LIN {X 0.280,Y -585.042,Z 449.322,A 0.000,B 0.000,C 90.000,E1 93.898} C_DIS
LIN {X -0.262,Y -588.278,Z 449.321,A 0.000,B 0.000,C 90.000,E1 93.841} C_DIS
LIN {X 0.026,Y -594.266,Z 449.320,A 0.000,B 0.000,C 90.000,E1 93.555} C_DIS
LIN {X 0.139,Y -599.956,Z 449.318,A 0.000,B 0.000,C 90.000,E1 93.212} C_DIS
LIN {X 0.002,Y -602.192,Z 449.317,A 0.000,B 0.000,C 90.000,E1 93.037} C_DIS
LIN {X -0.130,Y -605.915,Z 449.315,A 0.000,B 0.000,C 90.000,E1 92.694} C_DIS
LIN {X -0.222,Y -607.048,Z 449.314,A 0.000,B 0.000,C 90.000,E1 92.579} C_DIS
LIN {X 0.213,Y -608.066,Z 449.314,A 0.000,B 0.000,C 90.000,E1 92.407} C_DIS
LIN {X 0.153,Y -611.379,Z 449.311,A 0.000,B 0.000,C 90.000,E1 91.892} C_DIS
LIN {X 0.008,Y -612.023,Z 449.310,A 0.000,B 0.000,C 90.000,E1 91.776} C_DIS
LIN {X -0.029,Y -613.760,Z 449.307,A 0.000,B 0.000,C 90.000,E1 91.260} C_DIS
LIN {X -0.053,Y -614.433,Z 449.304,A 0.000,B 0.000,C 90.000,E1 90.745} C_DIS
LIN {X -0.069,Y -614.364,Z 449.301,A 0.000,B 0.000,C 90.000,E1 90.229} C_DIS
LIN {X 0.230,Y -614.158,Z 449.300,A 0.000,B 0.000,C 90.000,E1 89.943} C_DIS
LIN {X 0.214,Y -613.214,Z 449.297,A 0.000,B 0.000,C 90.000,E1 89.427} C_DIS
LIN {X -0.103,Y -612.227,Z 449.296,A 0.000,B 0.000,C 90.000,E1 89.198} C_DIS
LIN {X 0.030,Y -610.434,Z 449.293,A 0.000,B 0.000,C 90.000,E1 88.797} C_DIS
LIN {X -0.293,Y -608.948,Z 449.292,A 0.000,B 0.000,C 90.000,E1 88.568} C_DIS
LIN {X -0.015,Y -607.715,Z 449.290,A 0.000,B 0.000,C 90.000,E1 88.282} C_DIS
LIN {X 0.278,Y -606.083,Z 449.289,A 0.000,B 0.000,C 90.000,E1 87.993} C_DIS
LIN {X -0.227,Y -602.821,Z 449.287,A 0.000,B 0.000,C 90.000,E1 87.650} C_DIS
LIN {X 0.202,Y -601.337,Z 449.286,A 0.000,B 0.000,C 90.000,E1 87.478} C_DIS
LIN {X 0.029,Y -600.076,Z 449.285,A 0.000,B 0.000,C 90.000,E1 87.364} C_DIS
LIN {X 0.231,Y -595.856,Z 449.284,A 0.000,B 0.000,C 90.000,E1 87.020} C_DIS
LIN {X -0.293,Y -594.342,Z 449.283,A 0.000,B 0.000,C 90.000,E1 86.963} C_DIS
LIN {X -0.169,Y -592.394,Z 449.282,A 0.000,B 0.000,C 90.000,E1 86.846} C_DIS
LIN {X 0.126,Y -586.734,Z 449.281,A 0.000,B 0.000,C 90.000,E1 86.560} C_DIS
LIN {X 0.217,Y -581.356,Z 449.280,A 0.000,B 0.000,C 90.000,E1 86.331} C_DIS
LIN {X 0.124,Y -575.212,Z 449.279,A 0.000,B 0.000,C 90.000,E1 86.159} C_DIS
LIN {X -0.058,Y -574.482,Z 449.279,A 0.000,B 0.000,C 90.000,E1 86.159} C_DIS
LIN {X 0.129,Y -568.949,Z 449.278,A 0.000,B 0.000,C 90.000,E1 86.102} C_DIS
LIN {X 0.017,Y -568.335,Z 449.278,A 0.000,B 0.000,C 90.000,E1 86.102} C_DIS
LIN {X -0.038,Y -564.720,Z 449.278,A 0.000,B 0.000,C 90.000,E1 86.102} C_DIS
LIN {X -0.081,Y -486.304,Z 449.278,A 0.000,B 0.000,C 90.000,E1 86.102} C_DIS
LIN {X -0.033,Y -484.694,Z 449.254,A 0.000,B 0.000,C 90.000,E1 81.781} C_DIS
LIN {X -0.164,Y -484.577,Z 449.253,A 0.000,B 0.000,C 90.000,E1 81.489} C_DIS
LIN {X 0.184,Y -480.515,Z 449.227,A 0.000,B 0.000,C 90.000,E1 76.825} C_DIS
LIN {X 0.080,Y -474.266,Z 449.201,A 0.000,B 0.000,C 90.000,E1 72.181} C_DIS
LIN {X 0.048,Y -473.808,Z 449.199,A 0.000,B 0.000,C 90.000,E1 71.873} C_DIS
LIN {X 0.009,Y -466.228,Z 449.175,A 0.000,B 0.000,C 90.000,E1 67.486} C_DIS
LIN {X -0.049,Y -465.800,Z 449.173,A 0.000,B 0.000,C 90.000,E1 67.177} C_DIS
LIN {X 0.013,Y -464.449,Z 449.170,A 0.000,B 0.000,C 90.000,E1 66.538} C_DIS
LIN {X 0.209,Y -460.828,Z 449.160,A 0.000,B 0.000,C 90.000,E1 64.845} C_DIS
LIN {X 0.170,Y -460.829,Z 449.160,A 0.000,B 0.000,C 90.000,E1 64.845} C_DIS
LIN {X -0.103,Y -471.322,Z 449.152,A 0.000,B 0.000,C 90.000,E1 63.384} C_DIS
LIN {X -0.221,Y -476.895,Z 449.148,A 0.000,B 0.000,C 90.000,E1 62.615} C_DIS
LIN {X -0.218,Y -485.100,Z 449.141,A 0.000,B 0.000,C 90.000,E1 61.385} C_DIS
LIN {X 0.023,Y -489.694,Z 449.137,A 0.000,B 0.000,C 90.000,E1 60.589} C_DIS
LIN {X -0.151,Y -493.132,Z 449.133,A 0.000,B 0.000,C 90.000,E1 59.999} C_DIS
LIN {X -0.096,Y -495.546,Z 449.131,A 0.000,B 0.000,C 90.000,E1 59.537} C_DIS
LIN {X -0.176,Y -499.043,Z 449.127,A 0.000,B 0.000,C 90.000,E1 58.791} C_DIS
LIN {X -0.288,Y -501.495,Z 449.123,A 0.000,B 0.000,C 90.000,E1 58.201} C_DIS
LIN {X -0.118,Y -503.559,Z 449.120,A 0.000,B 0.000,C 90.000,E1 57.582} C_DIS
LIN {X -0.320,Y -506.063,Z 449.115,A 0.000,B 0.000,C 90.000,E1 56.707} C_DIS
LIN {X -0.116,Y -507.415,Z 449.112,A 0.000,B 0.000,C 90.000,E1 56.087} C_DIS
LIN {X 0.004,Y -508.918,Z 449.107,A 0.000,B 0.000,C 90.000,E1 55.182} C_DIS
LIN {X 0.139,Y -509.898,Z 449.102,A 0.000,B 0.000,C 90.000,E1 54.276} C_DIS
LIN {X -0.128,Y -510.426,Z 449.097,A 0.000,B 0.000,C 90.000,E1 53.417} C_DIS
LIN {X 0.242,Y -510.681,Z 449.090,A 0.000,B 0.000,C 90.000,E1 52.190} C_DIS
LIN {X 0.069,Y -510.714,Z 449.087,A 0.000,B 0.000,C 90.000,E1 51.618} C_DIS
LIN {X 0.040,Y -510.361,Z 449.080,A 0.000,B 0.000,C 90.000,E1 50.436} C_DIS
LIN {X 0.095,Y -509.924,Z 449.075,A 0.000,B 0.000,C 90.000,E1 49.542} C_DIS
LIN {X -0.099,Y -508.911,Z 449.067,A 0.000,B 0.000,C 90.000,E1 48.081} C_DIS
LIN {X -0.202,Y -507.992,Z 449.061,A 0.000,B 0.000,C 90.000,E1 46.905} C_DIS
LIN {X -0.318,Y -506.955,Z 449.054,A 0.000,B 0.000,C 90.000,E1 45.729} C_DIS
LIN {X -0.126,Y -505.056,Z 449.042,A 0.000,B 0.000,C 90.000,E1 43.623} C_DIS
LIN {X -0.190,Y -503.451,Z 449.032,A 0.000,B 0.000,C 90.000,E1 41.838} C_DIS
LIN {X -0.120,Y -502.051,Z 449.024,A 0.000,B 0.000,C 90.000,E1 40.334} C_DIS
LIN {X -0.076,Y -500.610,Z 449.016,A 0.000,B 0.000,C 90.000,E1 38.830} C_DIS
LIN {X 0.140,Y -499.520,Z 449.009,A 0.000,B 0.000,C 90.000,E1 37.604} C_DIS
LIN {X 0.083,Y -497.644,Z 448.999,A 0.000,B 0.000,C 90.000,E1 35.804} C_DIS
LIN {X 0.093,Y -495.608,Z 448.989,A 0.000,B 0.000,C 90.000,E1 33.992} C_DIS
LIN {X -0.070,Y -494.119,Z 448.982,A 0.000,B 0.000,C 90.000,E1 32.801} C_DIS
LIN {X -0.264,Y -491.817,Z 448.972,A 0.000,B 0.000,C 90.000,E1 31.003} C_DIS
LIN {X 0.091,Y -490.273,Z 448.965,A 0.000,B 0.000,C 90.000,E1 29.745} C_DIS
LIN {X -0.186,Y -487.521,Z 448.953,A 0.000,B 0.000,C 90.000,E1 27.641} C_DIS
LIN {X 0.105,Y -484.639,Z 448.940,A 0.000,B 0.000,C 90.000,E1 25.155} C_DIS
LIN {X 0.102,Y -481.751,Z 448.923,A 0.000,B 0.000,C 90.000,E1 22.078} C_DIS
LIN {X -0.089,Y -480.184,Z 448.911,A 0.000,B 0.000,C 90.000,E1 19.939} C_DIS
LIN {X 0.145,Y -479.024,Z 448.900,A 0.000,B 0.000,C 90.000,E1 18.055} C_DIS
LIN {X 0.056,Y -477.797,Z 448.890,A 0.000,B 0.000,C 90.000,E1 16.205} C_DIS
LIN {X -0.020,Y -476.715,Z 448.882,A 0.000,B 0.000,C 90.000,E1 14.662} C_DIS
LIN {X -0.033,Y -475.299,Z 448.868,A 0.000,B 0.000,C 90.000,E1 12.175} C_DIS
LIN {X 0.065,Y -474.352,Z 448.854,A 0.000,B 0.000,C 90.000,E1 9.670} C_DIS
LIN {X -0.039,Y -474.103,Z 448.849,A 0.000,B 0.000,C 90.000,E1 8.746} C_DIS
LIN {X -0.156,Y -473.933,Z 448.826,A 0.000,B 0.000,C 90.000,E1 4.702} C_DIS
LIN {X -0.023,Y -475.423,Z 448.804,A 0.000,B 0.000,C 90.000,E1 0.630} C_DIS
LIN {X -0.013,Y -477.940,Z 448.785,A 0.000,B 0.000,C 90.000,E1 357.306} C_DIS
LIN {X -0.097,Y -480.676,Z 448.771,A 0.000,B 0.000,C 90.000,E1 354.837} C_DIS
LIN {X 0.000,Y -483.958,Z 448.758,A 0.000,B 0.000,C 90.000,E1 352.356} C_DIS
LIN {X -0.018,Y -487.182,Z 448.746,A 0.000,B 0.000,C 90.000,E1 350.208} C_DIS
LIN {X -0.090,Y -495.576,Z 448.720,A 0.000,B 0.000,C 90.000,E1 345.644} C_DIS
LIN {X 0.146,Y -500.335,Z 448.708,A 0.000,B 0.000,C 90.000,E1 343.504} C_DIS
LIN {X -0.300,Y -506.989,Z 448.694,A 0.000,B 0.000,C 90.000,E1 340.859} C_DIS
LIN {X 0.233,Y -512.497,Z 448.682,A 0.000,B 0.000,C 90.000,E1 338.720} C_DIS
LIN {X -0.111,Y -516.460,Z 448.674,A 0.000,B 0.000,C 90.000,E1 337.283} C_DIS
LIN {X -0.087,Y -521.973,Z 448.662,A 0.000,B 0.000,C 90.000,E1 335.229} C_DIS
LIN {X 0.117,Y -526.692,Z 448.653,A 0.000,B 0.000,C 90.000,E1 333.461} C_DIS
LIN {X 0.014,Y -530.575,Z 448.645,A 0.000,B 0.000,C 90.000,E1 332.025} C_DIS
LIN {X -0.300,Y -535.330,Z 448.635,A 0.000,B 0.000,C 90.000,E1 330.333} C_DIS
LIN {X -0.153,Y -537.751,Z 448.630,A 0.000,B 0.000,C 90.000,E1 329.459} C_DIS
LIN {X -0.056,Y -542.540,Z 448.621,A 0.000,B 0.000,C 90.000,E1 327.740} C_DIS
LIN {X 0.228,Y -546.447,Z 448.613,A 0.000,B 0.000,C 90.000,E1 326.294} C_DIS
LIN {X 0.137,Y -550.354,Z 448.605,A 0.000,B 0.000,C 90.000,E1 324.895} C_DIS
LIN {X -0.111,Y -556.790,Z 448.593,A 0.000,B 0.000,C 90.000,E1 322.683} C_DIS
LIN {X 0.156,Y -563.379,Z 448.580,A 0.000,B 0.000,C 90.000,E1 320.436} C_DIS
LIN {X 0.295,Y -568.567,Z 448.571,A 0.000,B 0.000,C 90.000,E1 318.771} C_DIS
LIN {X -0.004,Y -572.710,Z 448.564,A 0.000,B 0.000,C 90.000,E1 317.433} C_DIS
LIN {X -0.096,Y -577.611,Z 448.555,A 0.000,B 0.000,C 90.000,E1 315.810} C_DIS
LIN {X -0.107,Y -582.531,Z 448.546,A 0.000,B 0.000,C 90.000,E1 314.190} C_DIS
LIN {X 0.151,Y -588.401,Z 448.535,A 0.000,B 0.000,C 90.000,E1 312.285} C_DIS
LIN {X -0.210,Y -592.519,Z 448.528,A 0.000,B 0.000,C 90.000,E1 310.987} C_DIS
LIN {X -0.049,Y -596.549,Z 448.520,A 0.000,B 0.000,C 90.000,E1 309.644} C_DIS
LIN {X 0.052,Y -601.175,Z 448.511,A 0.000,B 0.000,C 90.000,E1 308.051} C_DIS
LIN {X -0.006,Y -604.976,Z 448.504,A 0.000,B 0.000,C 90.000,E1 306.744} C_DIS
LIN {X -0.012,Y -608.601,Z 448.497,A 0.000,B 0.000,C 90.000,E1 305.438} C_DIS
LIN {X -0.035,Y -610.772,Z 448.493,A 0.000,B 0.000,C 90.000,E1 304.659} C_DIS
LIN {X -0.149,Y -614.195,Z 448.485,A 0.000,B 0.000,C 90.000,E1 303.372} C_DIS
LIN {X 0.104,Y -618.070,Z 448.477,A 0.000,B 0.000,C 90.000,E1 301.799} C_DIS
LIN {X 0.104,Y -621.763,Z 448.468,A 0.000,B 0.000,C 90.000,E1 300.256} C_DIS
LIN {X -0.144,Y -624.574,Z 448.461,A 0.000,B 0.000,C 90.000,E1 298.999} C_DIS
LIN {X -0.056,Y -628.494,Z 448.451,A 0.000,B 0.000,C 90.000,E1 297.206} C_DIS
LIN {X 0.044,Y -630.613,Z 448.446,A 0.000,B 0.000,C 90.000,E1 296.181} C_DIS
LIN {X 0.205,Y -633.127,Z 448.438,A 0.000,B 0.000,C 90.000,E1 294.899} C_DIS
LIN {X 0.176,Y -635.790,Z 448.430,A 0.000,B 0.000,C 90.000,E1 293.387} C_DIS
LIN {X -0.058,Y -638.246,Z 448.422,A 0.000,B 0.000,C 90.000,E1 291.897} C_DIS
LIN {X 0.299,Y -640.073,Z 448.415,A 0.000,B 0.000,C 90.000,E1 290.610} C_DIS
LIN {X 0.038,Y -641.527,Z 448.409,A 0.000,B 0.000,C 90.000,E1 289.631} C_DIS
LIN {X -0.212,Y -642.795,Z 448.404,A 0.000,B 0.000,C 90.000,E1 288.652} C_DIS
LIN {X -0.196,Y -644.148,Z 448.397,A 0.000,B 0.000,C 90.000,E1 287.402} C_DIS
LIN {X -0.111,Y -645.549,Z 448.388,A 0.000,B 0.000,C 90.000,E1 285.898} C_DIS
LIN {X -0.066,Y -646.361,Z 448.383,A 0.000,B 0.000,C 90.000,E1 284.898} C_DIS
LIN {X 0.015,Y -647.149,Z 448.376,A 0.000,B 0.000,C 90.000,E1 283.647} C_DIS
LIN {X 0.085,Y -647.640,Z 448.370,A 0.000,B 0.000,C 90.000,E1 282.647} C_DIS
LIN {X -0.112,Y -648.117,Z 448.363,A 0.000,B 0.000,C 90.000,E1 281.422} C_DIS
LIN {X -0.038,Y -648.313,Z 448.358,A 0.000,B 0.000,C 90.000,E1 280.423} C_DIS
LIN {X -0.338,Y -648.217,Z 448.351,A 0.000,B 0.000,C 90.000,E1 279.208} C_DIS
LIN {X -0.237,Y -648.029,Z 448.347,A 0.000,B 0.000,C 90.000,E1 278.454} C_DIS
LIN {X 0.110,Y -647.485,Z 448.340,A 0.000,B 0.000,C 90.000,E1 277.182} C_DIS
LIN {X 0.197,Y -647.015,Z 448.336,A 0.000,B 0.000,C 90.000,E1 276.429} C_DIS
LIN {X 0.205,Y -646.363,Z 448.332,A 0.000,B 0.000,C 90.000,E1 275.682} C_DIS
LIN {X 0.036,Y -645.158,Z 448.326,A 0.000,B 0.000,C 90.000,E1 274.702} C_DIS
LIN {X 0.028,Y -644.107,Z 448.322,A 0.000,B 0.000,C 90.000,E1 273.955} C_DIS
LIN {X -0.228,Y -642.506,Z 448.316,A 0.000,B 0.000,C 90.000,E1 272.980} C_DIS
LIN {X -0.104,Y -640.224,Z 448.310,A 0.000,B 0.000,C 90.000,E1 271.718} C_DIS
LIN {X 0.209,Y -638.223,Z 448.304,A 0.000,B 0.000,C 90.000,E1 270.688} C_DIS
LIN {X -0.004,Y -634.937,Z 448.296,A 0.000,B 0.000,C 90.000,E1 269.198} C_DIS
LIN {X 0.235,Y -632.504,Z 448.290,A 0.000,B 0.000,C 90.000,E1 268.167} C_DIS
LIN {X 0.185,Y -629.317,Z 448.283,A 0.000,B 0.000,C 90.000,E1 266.906} C_DIS
LIN {X -0.161,Y -625.337,Z 448.274,A 0.000,B 0.000,C 90.000,E1 265.412} C_DIS
LIN {X 0.098,Y -621.272,Z 448.266,A 0.000,B 0.000,C 90.000,E1 263.856} C_DIS
LIN {X 0.227,Y -618.487,Z 448.260,A 0.000,B 0.000,C 90.000,E1 262.818} C_DIS
LIN {X -0.181,Y -614.200,Z 448.252,A 0.000,B 0.000,C 90.000,E1 261.310} C_DIS
LIN {X 0.186,Y -610.466,Z 448.245,A 0.000,B 0.000,C 90.000,E1 259.982} C_DIS
LIN {X -0.020,Y -606.615,Z 448.237,A 0.000,B 0.000,C 90.000,E1 258.701} C_DIS
LIN {X -0.169,Y -602.656,Z 448.230,A 0.000,B 0.000,C 90.000,E1 257.409} C_DIS
LIN {X 0.202,Y -598.611,Z 448.223,A 0.000,B 0.000,C 90.000,E1 256.061} C_DIS
LIN {X 0.070,Y -596.121,Z 448.218,A 0.000,B 0.000,C 90.000,E1 255.283} C_DIS
LIN {X -0.104,Y -591.867,Z 448.211,A 0.000,B 0.000,C 90.000,E1 253.976} C_DIS
LIN {X -0.182,Y -587.539,Z 448.204,A 0.000,B 0.000,C 90.000,E1 252.653} C_DIS
LIN {X 0.222,Y -583.092,Z 448.196,A 0.000,B 0.000,C 90.000,E1 251.275} C_DIS
LIN {X -0.212,Y -579.432,Z 448.190,A 0.000,B 0.000,C 90.000,E1 250.242} C_DIS
LIN {X 0.048,Y -575.781,Z 448.184,A 0.000,B 0.000,C 90.000,E1 249.135} C_DIS
LIN {X -0.126,Y -570.969,Z 448.177,A 0.000,B 0.000,C 90.000,E1 247.794} C_DIS
LIN {X 0.227,Y -566.950,Z 448.171,A 0.000,B 0.000,C 90.000,E1 246.666} C_DIS
LIN {X 0.098,Y -561.760,Z 448.163,A 0.000,B 0.000,C 90.000,E1 245.305} C_DIS
LIN {X 0.131,Y -555.431,Z 448.154,A 0.000,B 0.000,C 90.000,E1 243.640} C_DIS
LIN {X 0.033,Y -549.002,Z 448.144,A 0.000,B 0.000,C 90.000,E1 241.975} C_DIS
LIN {X 0.059,Y -541.652,Z 448.133,A 0.000,B 0.000,C 90.000,E1 239.999} C_DIS
LIN {X 0.177,Y -534.469,Z 448.122,A 0.000,B 0.000,C 90.000,E1 237.995} C_DIS
LIN {X -0.032,Y -528.228,Z 448.113,A 0.000,B 0.000,C 90.000,E1 236.294} C_DIS
LIN {X -0.084,Y -522.049,Z 448.103,A 0.000,B 0.000,C 90.000,E1 234.562} C_DIS
LIN {X 0.271,Y -514.861,Z 448.092,A 0.000,B 0.000,C 90.000,E1 232.477} C_DIS
LIN {X 0.068,Y -505.494,Z 448.075,A 0.000,B 0.000,C 90.000,E1 229.542} C_DIS
LIN {X -0.217,Y -501.066,Z 448.067,A 0.000,B 0.000,C 90.000,E1 228.081} C_DIS
LIN {X 0.123,Y -496.709,Z 448.059,A 0.000,B 0.000,C 90.000,E1 226.539} C_DIS
LIN {X 0.184,Y -489.920,Z 448.045,A 0.000,B 0.000,C 90.000,E1 224.109} C_DIS
LIN {X 0.100,Y -485.033,Z 448.035,A 0.000,B 0.000,C 90.000,E1 222.285} C_DIS
LIN {X -0.061,Y -480.269,Z 448.025,A 0.000,B 0.000,C 90.000,E1 220.458} C_DIS
LIN {X -0.172,Y -474.944,Z 448.013,A 0.000,B 0.000,C 90.000,E1 218.302} C_DIS
LIN {X -0.034,Y -468.523,Z 447.997,A 0.000,B 0.000,C 90.000,E1 215.471} C_DIS
LIN {X -0.023,Y -464.476,Z 447.987,A 0.000,B 0.000,C 90.000,E1 213.579} C_DIS
LIN {X -0.122,Y -459.209,Z 447.972,A 0.000,B 0.000,C 90.000,E1 211.052} C_DIS
LIN {X -0.165,Y -456.005,Z 447.964,A 0.000,B 0.000,C 90.000,E1 209.461} C_DIS
LIN {X -0.090,Y -452.779,Z 447.955,A 0.000,B 0.000,C 90.000,E1 207.847} C_DIS
LIN {X -0.074,Y -449.527,Z 447.946,A 0.000,B 0.000,C 90.000,E1 206.232} C_DIS
LIN {X 0.000,Y -444.815,Z 447.933,A 0.000,B 0.000,C 90.000,E1 203.951} C_DIS
LIN {X 0.147,Y -440.894,Z 447.922,A 0.000,B 0.000,C 90.000,E1 201.972} C_DIS
LIN {X 0.032,Y -436.381,Z 447.909,A 0.000,B 0.000,C 90.000,E1 199.685} C_DIS
LIN {X -0.005,Y -431.687,Z 447.895,A 0.000,B 0.000,C 90.000,E1 197.040} C_DIS
LIN {X 0.223,Y -428.444,Z 447.884,A 0.000,B 0.000,C 90.000,E1 195.009} C_DIS
LIN {X -0.077,Y -424.908,Z 447.871,A 0.000,B 0.000,C 90.000,E1 192.703} C_DIS
LIN {X -0.023,Y -420.328,Z 447.852,A 0.000,B 0.000,C 90.000,E1 189.321} C_DIS
LIN {X -0.100,Y -417.898,Z 447.841,A 0.000,B 0.000,C 90.000,E1 187.296} C_DIS
LIN {X 0.179,Y -415.008,Z 447.825,A 0.000,B 0.000,C 90.000,E1 184.531} C_DIS
LIN {X -0.133,Y -412.454,Z 447.810,A 0.000,B 0.000,C 90.000,E1 181.835} C_DIS
LIN {X -0.124,Y -410.004,Z 447.789,A 0.000,B 0.000,C 90.000,E1 178.051} C_DIS
LIN {X -0.144,Y -408.668,Z 447.766,A 0.000,B 0.000,C 90.000,E1 173.913} C_DIS
LIN {X -0.059,Y -408.839,Z 447.749,A 0.000,B 0.000,C 90.000,E1 170.792} C_DIS
LIN {X -0.040,Y -410.037,Z 447.728,A 0.000,B 0.000,C 90.000,E1 166.992} C_DIS
LIN {X -0.110,Y -412.024,Z 447.709,A 0.000,B 0.000,C 90.000,E1 163.559} C_DIS
LIN {X -0.013,Y -415.002,Z 447.690,A 0.000,B 0.000,C 90.000,E1 160.115} C_DIS
LIN {X 0.099,Y -417.197,Z 447.678,A 0.000,B 0.000,C 90.000,E1 158.050} C_DIS
LIN {X 0.223,Y -421.074,Z 447.661,A 0.000,B 0.000,C 90.000,E1 154.973} C_DIS
LIN {X 0.158,Y -424.385,Z 447.648,A 0.000,B 0.000,C 90.000,E1 152.615} C_DIS
LIN {X 0.204,Y -427.985,Z 447.635,A 0.000,B 0.000,C 90.000,E1 150.255} C_DIS
LIN {X -0.033,Y -430.105,Z 447.628,A 0.000,B 0.000,C 90.000,E1 148.948} C_DIS
LIN {X -0.100,Y -435.215,Z 447.611,A 0.000,B 0.000,C 90.000,E1 145.960} C_DIS
LIN {X 0.110,Y -440.091,Z 447.596,A 0.000,B 0.000,C 90.000,E1 143.290} C_DIS
LIN {X 0.052,Y -442.701,Z 447.589,A 0.000,B 0.000,C 90.000,E1 141.984} C_DIS
LIN {X 0.006,Y -446.040,Z 447.580,A 0.000,B 0.000,C 90.000,E1 140.356} C_DIS
LIN {X 0.020,Y -449.451,Z 447.571,A 0.000,B 0.000,C 90.000,E1 138.728} C_DIS
LIN {X -0.286,Y -452.143,Z 447.564,A 0.000,B 0.000,C 90.000,E1 137.472} C_DIS
LIN {X 0.113,Y -455.291,Z 447.555,A 0.000,B 0.000,C 90.000,E1 135.810} C_DIS
LIN {X 0.188,Y -456.958,Z 447.549,A 0.000,B 0.000,C 90.000,E1 134.838} C_DIS
LIN {X 0.283,Y -458.534,Z 447.544,A 0.000,B 0.000,C 90.000,E1 133.866} C_DIS
LIN {X 0.117,Y -460.215,Z 447.537,A 0.000,B 0.000,C 90.000,E1 132.609} C_DIS
LIN {X -0.028,Y -461.379,Z 447.530,A 0.000,B 0.000,C 90.000,E1 131.353} C_DIS
LIN {X 0.142,Y -461.921,Z 447.524,A 0.000,B 0.000,C 90.000,E1 130.378} C_DIS
LIN {X 0.025,Y -461.985,Z 447.519,A 0.000,B 0.000,C 90.000,E1 129.439} C_DIS
LIN {X -0.190,Y -461.777,Z 447.516,A 0.000,B 0.000,C 90.000,E1 128.830} C_DIS
LIN {X -0.019,Y -461.057,Z 447.510,A 0.000,B 0.000,C 90.000,E1 127.855} C_DIS
LIN {X 0.225,Y -459.977,Z 447.505,A 0.000,B 0.000,C 90.000,E1 126.870} C_DIS
LIN {X 0.079,Y -459.118,Z 447.501,A 0.000,B 0.000,C 90.000,E1 126.251} C_DIS
LIN {X 0.200,Y -458.102,Z 447.498,A 0.000,B 0.000,C 90.000,E1 125.598} C_DIS
LIN {X 0.038,Y -456.132,Z 447.493,A 0.000,B 0.000,C 90.000,E1 124.659} C_DIS
LIN {X -0.132,Y -454.724,Z 447.489,A 0.000,B 0.000,C 90.000,E1 124.040} C_DIS
LIN {X -0.123,Y -451.310,Z 447.482,A 0.000,B 0.000,C 90.000,E1 122.752} C_DIS
LIN {X 0.139,Y -448.558,Z 447.477,A 0.000,B 0.000,C 90.000,E1 121.750} C_DIS
LIN {X -0.013,Y -445.715,Z 447.471,A 0.000,B 0.000,C 90.000,E1 120.797} C_DIS
LIN {X 0.069,Y -440.549,Z 447.462,A 0.000,B 0.000,C 90.000,E1 119.155} C_DIS
LIN {X 0.105,Y -436.433,Z 447.455,A 0.000,B 0.000,C 90.000,E1 117.897} C_DIS
LIN {X 0.066,Y -436.421,Z 447.455,A 0.000,B 0.000,C 90.000,E1 117.897} C_DIS
LIN {X -0.083,Y -444.882,Z 447.438,A 0.000,B 0.000,C 90.000,E1 114.899} C_DIS
LIN {X 0.176,Y -453.993,Z 447.417,A 0.000,B 0.000,C 90.000,E1 110.972} C_DIS
LIN {X 0.288,Y -456.641,Z 447.411,A 0.000,B 0.000,C 90.000,E1 109.993} C_DIS
LIN {X 0.035,Y -457.454,Z 447.410,A 0.000,B 0.000,C 90.000,E1 109.704} C_DIS
LIN {X 0.136,Y -466.113,Z 447.387,A 0.000,B 0.000,C 90.000,E1 105.552} C_DIS
LIN {X -0.140,Y -467.684,Z 447.383,A 0.000,B 0.000,C 90.000,E1 104.954} C_DIS
LIN {X -0.183,Y -475.897,Z 447.357,A 0.000,B 0.000,C 90.000,E1 100.254} C_DIS
LIN {X 0.124,Y -476.347,Z 447.355,A 0.000,B 0.000,C 90.000,E1 99.905} C_DIS
LIN {X 0.081,Y -481.861,Z 447.331,A 0.000,B 0.000,C 90.000,E1 95.568} C_DIS
LIN {X -0.072,Y -482.189,Z 447.329,A 0.000,B 0.000,C 90.000,E1 95.277} C_DIS
LIN {X -0.196,Y -483.242,Z 447.319,A 0.000,B 0.000,C 90.000,E1 93.383} C_DIS
LIN {X -0.266,Y -574.386,Z 447.319,A 0.000,B 0.000,C 90.000,E1 93.383} C_DIS
LIN {X -0.113,Y -580.591,Z 447.318,A 0.000,B 0.000,C 90.000,E1 93.326} C_DIS
LIN {X -0.167,Y -585.370,Z 447.318,A 0.000,B 0.000,C 90.000,E1 93.212} C_DIS
LIN {X 0.174,Y -587.515,Z 447.317,A 0.000,B 0.000,C 90.000,E1 93.094} C_DIS
LIN {X -0.154,Y -593.010,Z 447.316,A 0.000,B 0.000,C 90.000,E1 92.808} C_DIS
LIN {X -0.270,Y -595.548,Z 447.315,A 0.000,B 0.000,C 90.000,E1 92.636} C_DIS
LIN {X -0.103,Y -597.917,Z 447.313,A 0.000,B 0.000,C 90.000,E1 92.407} C_DIS
LIN {X -0.171,Y -599.097,Z 447.313,A 0.000,B 0.000,C 90.000,E1 92.293} C_DIS
LIN {X 0.002,Y -601.982,Z 447.311,A 0.000,B 0.000,C 90.000,E1 91.892} C_DIS
LIN {X -0.083,Y -604.590,Z 447.308,A 0.000,B 0.000,C 90.000,E1 91.375} C_DIS
LIN {X 0.175,Y -605.465,Z 447.306,A 0.000,B 0.000,C 90.000,E1 91.088} C_DIS
LIN {X -0.168,Y -606.018,Z 447.305,A 0.000,B 0.000,C 90.000,E1 90.859} C_DIS
LIN {X 0.096,Y -606.343,Z 447.303,A 0.000,B 0.000,C 90.000,E1 90.573} C_DIS
LIN {X 0.026,Y -606.295,Z 447.300,A 0.000,B 0.000,C 90.000,E1 90.057} C_DIS
LIN {X -0.044,Y -605.152,Z 447.297,A 0.000,B 0.000,C 90.000,E1 89.542} C_DIS
LIN {X 0.221,Y -604.220,Z 447.296,A 0.000,B 0.000,C 90.000,E1 89.255} C_DIS
LIN {X -0.291,Y -602.491,Z 447.294,A 0.000,B 0.000,C 90.000,E1 88.912} C_DIS
LIN {X 0.212,Y -599.532,Z 447.291,A 0.000,B 0.000,C 90.000,E1 88.339} C_DIS
LIN {X 0.035,Y -598.547,Z 447.290,A 0.000,B 0.000,C 90.000,E1 88.224} C_DIS
LIN {X 0.261,Y -592.687,Z 447.287,A 0.000,B 0.000,C 90.000,E1 87.707} C_DIS
LIN {X 0.266,Y -589.284,Z 447.286,A 0.000,B 0.000,C 90.000,E1 87.478} C_DIS
LIN {X -0.185,Y -587.477,Z 447.286,A 0.000,B 0.000,C 90.000,E1 87.421} C_DIS
LIN {X -0.268,Y -583.534,Z 447.285,A 0.000,B 0.000,C 90.000,E1 87.249} C_DIS
LIN {X 0.094,Y -581.560,Z 447.284,A 0.000,B 0.000,C 90.000,E1 87.135} C_DIS
LIN {X -0.016,Y -579.378,Z 447.284,A 0.000,B 0.000,C 90.000,E1 87.078} C_DIS
LIN {X 0.023,Y -575.162,Z 447.283,A 0.000,B 0.000,C 90.000,E1 86.963} C_DIS
LIN {X 0.172,Y -572.267,Z 447.283,A 0.000,B 0.000,C 90.000,E1 86.906} C_DIS
LIN {X -0.051,Y -568.057,Z 447.283,A 0.000,B 0.000,C 90.000,E1 86.906} C_DIS
LIN {X -0.092,Y -486.228,Z 447.283,A 0.000,B 0.000,C 90.000,E1 86.906} C_DIS
LIN {X 0.017,Y -486.385,Z 447.281,A 0.000,B 0.000,C 90.000,E1 86.560} C_DIS
LIN {X -0.158,Y -486.365,Z 447.279,A 0.000,B 0.000,C 90.000,E1 86.274} C_DIS
LIN {X -0.070,Y -484.690,Z 447.254,A 0.000,B 0.000,C 90.000,E1 81.659} C_DIS
LIN {X 0.076,Y -484.059,Z 447.250,A 0.000,B 0.000,C 90.000,E1 81.027} C_DIS
LIN {X -0.160,Y -480.632,Z 447.228,A 0.000,B 0.000,C 90.000,E1 77.048} C_DIS
LIN {X 0.166,Y -480.324,Z 447.226,A 0.000,B 0.000,C 90.000,E1 76.700} C_DIS
LIN {X 0.071,Y -474.138,Z 447.200,A 0.000,B 0.000,C 90.000,E1 72.054} C_DIS
LIN {X -0.063,Y -465.611,Z 447.173,A 0.000,B 0.000,C 90.000,E1 67.050} C_DIS
LIN {X -0.064,Y -461.284,Z 447.162,A 0.000,B 0.000,C 90.000,E1 65.101} C_DIS
LIN {X -0.104,Y -461.293,Z 447.162,A 0.000,B 0.000,C 90.000,E1 65.101} C_DIS
LIN {X -0.116,Y -472.021,Z 447.153,A 0.000,B 0.000,C 90.000,E1 63.589} C_DIS
LIN {X 0.183,Y -478.633,Z 447.148,A 0.000,B 0.000,C 90.000,E1 62.615} C_DIS
LIN {X 0.033,Y -485.877,Z 447.142,A 0.000,B 0.000,C 90.000,E1 61.563} C_DIS
LIN {X 0.048,Y -490.561,Z 447.138,A 0.000,B 0.000,C 90.000,E1 60.795} C_DIS
LIN {X -0.120,Y -494.070,Z 447.134,A 0.000,B 0.000,C 90.000,E1 60.205} C_DIS
LIN {X -0.014,Y -497.249,Z 447.131,A 0.000,B 0.000,C 90.000,E1 59.587} C_DIS
LIN {X -0.135,Y -500.098,Z 447.128,A 0.000,B 0.000,C 90.000,E1 58.997} C_DIS
LIN {X -0.237,Y -502.582,Z 447.124,A 0.000,B 0.000,C 90.000,E1 58.408} C_DIS
LIN {X -0.061,Y -504.728,Z 447.121,A 0.000,B 0.000,C 90.000,E1 57.788} C_DIS
LIN {X 0.134,Y -506.495,Z 447.118,A 0.000,B 0.000,C 90.000,E1 57.168} C_DIS
LIN {X -0.250,Y -507.330,Z 447.116,A 0.000,B 0.000,C 90.000,E1 56.914} C_DIS
LIN {X -0.035,Y -508.712,Z 447.113,A 0.000,B 0.000,C 90.000,E1 56.294} C_DIS
LIN {X 0.192,Y -509.817,Z 447.109,A 0.000,B 0.000,C 90.000,E1 55.674} C_DIS
LIN {X 0.008,Y -510.673,Z 447.106,A 0.000,B 0.000,C 90.000,E1 55.102} C_DIS
LIN {X 0.252,Y -511.353,Z 447.103,A 0.000,B 0.000,C 90.000,E1 54.482} C_DIS
LIN {X 0.001,Y -511.945,Z 447.098,A 0.000,B 0.000,C 90.000,E1 53.623} C_DIS
LIN {X 0.083,Y -512.152,Z 447.091,A 0.000,B 0.000,C 90.000,E1 52.431} C_DIS
LIN {X 0.236,Y -512.214,Z 447.088,A 0.000,B 0.000,C 90.000,E1 51.823} C_DIS
LIN {X 0.231,Y -511.850,Z 447.082,A 0.000,B 0.000,C 90.000,E1 50.642} C_DIS
LIN {X -0.024,Y -511.415,Z 447.077,A 0.000,B 0.000,C 90.000,E1 49.784} C_DIS
LIN {X -0.196,Y -510.353,Z 447.068,A 0.000,B 0.000,C 90.000,E1 48.324} C_DIS
LIN {X -0.036,Y -509.136,Z 447.060,A 0.000,B 0.000,C 90.000,E1 46.824} C_DIS
LIN {X -0.137,Y -508.043,Z 447.054,A 0.000,B 0.000,C 90.000,E1 45.648} C_DIS
LIN {X -0.035,Y -505.795,Z 447.040,A 0.000,B 0.000,C 90.000,E1 43.257} C_DIS
LIN {X -0.076,Y -504.145,Z 447.030,A 0.000,B 0.000,C 90.000,E1 41.472} C_DIS
LIN {X 0.218,Y -502.426,Z 447.020,A 0.000,B 0.000,C 90.000,E1 39.644} C_DIS
LIN {X -0.170,Y -500.724,Z 447.010,A 0.000,B 0.000,C 90.000,E1 37.890} C_DIS
LIN {X -0.199,Y -498.871,Z 447.000,A 0.000,B 0.000,C 90.000,E1 36.091} C_DIS
LIN {X -0.159,Y -496.804,Z 446.990,A 0.000,B 0.000,C 90.000,E1 34.278} C_DIS
LIN {X 0.117,Y -495.352,Z 446.984,A 0.000,B 0.000,C 90.000,E1 33.038} C_DIS
LIN {X -0.204,Y -493.049,Z 446.974,A 0.000,B 0.000,C 90.000,E1 31.258} C_DIS
LIN {X -0.247,Y -491.076,Z 446.965,A 0.000,B 0.000,C 90.000,E1 29.745} C_DIS
LIN {X -0.068,Y -488.335,Z 446.953,A 0.000,B 0.000,C 90.000,E1 27.590} C_DIS
LIN {X -0.182,Y -485.467,Z 446.940,A 0.000,B 0.000,C 90.000,E1 25.155} C_DIS
LIN {X -0.154,Y -482.567,Z 446.923,A 0.000,B 0.000,C 90.000,E1 22.078} C_DIS
LIN {X 0.126,Y -480.821,Z 446.909,A 0.000,B 0.000,C 90.000,E1 19.577} C_DIS
LIN {X -0.068,Y -479.856,Z 446.900,A 0.000,B 0.000,C 90.000,E1 18.055} C_DIS
LIN {X -0.138,Y -478.605,Z 446.890,A 0.000,B 0.000,C 90.000,E1 16.205} C_DIS
LIN {X -0.077,Y -477.529,Z 446.881,A 0.000,B 0.000,C 90.000,E1 14.647} C_DIS
LIN {X -0.187,Y -476.089,Z 446.868,A 0.000,B 0.000,C 90.000,E1 12.175} C_DIS
LIN {X -0.065,Y -475.140,Z 446.854,A 0.000,B 0.000,C 90.000,E1 9.670} C_DIS
LIN {X -0.113,Y -474.600,Z 446.840,A 0.000,B 0.000,C 90.000,E1 7.182} C_DIS
LIN {X -0.163,Y -474.783,Z 446.823,A 0.000,B 0.000,C 90.000,E1 4.069} C_DIS
LIN {X -0.067,Y -476.157,Z 446.803,A 0.000,B 0.000,C 90.000,E1 0.630} C_DIS
LIN {X -0.193,Y -478.971,Z 446.783,A 0.000,B 0.000,C 90.000,E1 357.020} C_DIS
LIN {X -0.205,Y -481.808,Z 446.770,A 0.000,B 0.000,C 90.000,E1 354.546} C_DIS
LIN {X 0.068,Y -484.726,Z 446.758,A 0.000,B 0.000,C 90.000,E1 352.356} C_DIS
LIN {X 0.071,Y -487.981,Z 446.746,A 0.000,B 0.000,C 90.000,E1 350.208} C_DIS
LIN {X 0.146,Y -492.095,Z 446.732,A 0.000,B 0.000,C 90.000,E1 347.757} C_DIS
LIN {X 0.079,Y -497.048,Z 446.719,A 0.000,B 0.000,C 90.000,E1 345.338} C_DIS
LIN {X -0.193,Y -502.629,Z 446.705,A 0.000,B 0.000,C 90.000,E1 342.960} C_DIS
LIN {X 0.186,Y -510.194,Z 446.689,A 0.000,B 0.000,C 90.000,E1 339.934} C_DIS
LIN {X 0.090,Y -514.148,Z 446.680,A 0.000,B 0.000,C 90.000,E1 338.465} C_DIS
LIN {X -0.077,Y -517.359,Z 446.674,A 0.000,B 0.000,C 90.000,E1 337.305} C_DIS
LIN {X 0.172,Y -522.881,Z 446.663,A 0.000,B 0.000,C 90.000,E1 335.229} C_DIS
LIN {X -0.073,Y -527.632,Z 446.653,A 0.000,B 0.000,C 90.000,E1 333.512} C_DIS
LIN {X 0.317,Y -531.563,Z 446.645,A 0.000,B 0.000,C 90.000,E1 332.025} C_DIS
LIN {X 0.312,Y -535.543,Z 446.637,A 0.000,B 0.000,C 90.000,E1 330.589} C_DIS
LIN {X -0.092,Y -539.597,Z 446.629,A 0.000,B 0.000,C 90.000,E1 329.203} C_DIS
LIN {X -0.129,Y -544.431,Z 446.619,A 0.000,B 0.000,C 90.000,E1 327.502} C_DIS
LIN {X -0.059,Y -549.121,Z 446.610,A 0.000,B 0.000,C 90.000,E1 325.801} C_DIS
LIN {X -0.037,Y -553.872,Z 446.601,A 0.000,B 0.000,C 90.000,E1 324.116} C_DIS
LIN {X 0.079,Y -558.771,Z 446.591,A 0.000,B 0.000,C 90.000,E1 322.431} C_DIS
LIN {X -0.047,Y -565.416,Z 446.579,A 0.000,B 0.000,C 90.000,E1 320.231} C_DIS
LIN {X 0.127,Y -570.695,Z 446.570,A 0.000,B 0.000,C 90.000,E1 318.566} C_DIS
LIN {X -0.014,Y -575.665,Z 446.561,A 0.000,B 0.000,C 90.000,E1 316.944} C_DIS
LIN {X 0.204,Y -579.779,Z 446.553,A 0.000,B 0.000,C 90.000,E1 315.567} C_DIS
LIN {X -0.323,Y -583.938,Z 446.546,A 0.000,B 0.000,C 90.000,E1 314.271} C_DIS
LIN {X 0.160,Y -590.715,Z 446.534,A 0.000,B 0.000,C 90.000,E1 312.081} C_DIS
LIN {X -0.155,Y -594.829,Z 446.527,A 0.000,B 0.000,C 90.000,E1 310.782} C_DIS
LIN {X 0.051,Y -598.852,Z 446.519,A 0.000,B 0.000,C 90.000,E1 309.439} C_DIS
LIN {X 0.327,Y -602.748,Z 446.512,A 0.000,B 0.000,C 90.000,E1 308.096} C_DIS
LIN {X 0.290,Y -606.546,Z 446.505,A 0.000,B 0.000,C 90.000,E1 306.790} C_DIS
LIN {X -0.049,Y -610.246,Z 446.497,A 0.000,B 0.000,C 90.000,E1 305.518} C_DIS
LIN {X -0.054,Y -612.426,Z 446.493,A 0.000,B 0.000,C 90.000,E1 304.739} C_DIS
LIN {X -0.137,Y -615.873,Z 446.486,A 0.000,B 0.000,C 90.000,E1 303.452} C_DIS
LIN {X 0.157,Y -619.789,Z 446.477,A 0.000,B 0.000,C 90.000,E1 301.878} C_DIS
LIN {X 0.203,Y -622.900,Z 446.470,A 0.000,B 0.000,C 90.000,E1 300.590} C_DIS
LIN {X -0.029,Y -625.274,Z 446.464,A 0.000,B 0.000,C 90.000,E1 299.589} C_DIS
LIN {X 0.049,Y -628.627,Z 446.456,A 0.000,B 0.000,C 90.000,E1 298.052} C_DIS
LIN {X -0.093,Y -631.435,Z 446.449,A 0.000,B 0.000,C 90.000,E1 296.796} C_DIS
LIN {X 0.036,Y -633.500,Z 446.443,A 0.000,B 0.000,C 90.000,E1 295.771} C_DIS
LIN {X -0.077,Y -635.511,Z 446.438,A 0.000,B 0.000,C 90.000,E1 294.771} C_DIS
LIN {X -0.108,Y -637.796,Z 446.431,A 0.000,B 0.000,C 90.000,E1 293.515} C_DIS
LIN {X -0.160,Y -639.428,Z 446.425,A 0.000,B 0.000,C 90.000,E1 292.514} C_DIS
LIN {X 0.163,Y -641.047,Z 446.419,A 0.000,B 0.000,C 90.000,E1 291.482} C_DIS
LIN {X -0.140,Y -643.623,Z 446.410,A 0.000,B 0.000,C 90.000,E1 289.758} C_DIS
LIN {X 0.096,Y -645.199,Z 446.403,A 0.000,B 0.000,C 90.000,E1 288.489} C_DIS
LIN {X -0.110,Y -646.301,Z 446.397,A 0.000,B 0.000,C 90.000,E1 287.511} C_DIS
LIN {X -0.309,Y -647.940,Z 446.388,A 0.000,B 0.000,C 90.000,E1 285.788} C_DIS
LIN {X -0.196,Y -648.922,Z 446.381,A 0.000,B 0.000,C 90.000,E1 284.537} C_DIS
LIN {X 0.270,Y -649.708,Z 446.372,A 0.000,B 0.000,C 90.000,E1 283.008} C_DIS
LIN {X 0.246,Y -650.252,Z 446.366,A 0.000,B 0.000,C 90.000,E1 281.771} C_DIS
LIN {X 0.095,Y -650.474,Z 446.359,A 0.000,B 0.000,C 90.000,E1 280.546} C_DIS
LIN {X 0.081,Y -650.414,Z 446.353,A 0.000,B 0.000,C 90.000,E1 279.557} C_DIS
LIN {X 0.063,Y -650.245,Z 446.348,A 0.000,B 0.000,C 90.000,E1 278.568} C_DIS
LIN {X 0.211,Y -649.490,Z 446.339,A 0.000,B 0.000,C 90.000,E1 277.068} C_DIS
LIN {X 0.092,Y -648.739,Z 446.334,A 0.000,B 0.000,C 90.000,E1 276.087} C_DIS
LIN {X 0.185,Y -647.992,Z 446.330,A 0.000,B 0.000,C 90.000,E1 275.334} C_DIS
LIN {X -0.247,Y -646.369,Z 446.323,A 0.000,B 0.000,C 90.000,E1 274.131} C_DIS
LIN {X -0.014,Y -644.318,Z 446.316,A 0.000,B 0.000,C 90.000,E1 272.865} C_DIS
LIN {X -0.289,Y -642.541,Z 446.310,A 0.000,B 0.000,C 90.000,E1 271.892} C_DIS
LIN {X 0.077,Y -640.562,Z 446.305,A 0.000,B 0.000,C 90.000,E1 270.859} C_DIS
LIN {X -0.091,Y -637.263,Z 446.297,A 0.000,B 0.000,C 90.000,E1 269.370} C_DIS
LIN {X 0.182,Y -634.837,Z 446.291,A 0.000,B 0.000,C 90.000,E1 268.339} C_DIS
LIN {X -0.060,Y -630.915,Z 446.283,A 0.000,B 0.000,C 90.000,E1 266.846} C_DIS
LIN {X 0.215,Y -626.934,Z 446.274,A 0.000,B 0.000,C 90.000,E1 265.298} C_DIS
LIN {X 0.197,Y -622.141,Z 446.264,A 0.000,B 0.000,C 90.000,E1 263.514} C_DIS
LIN {X 0.031,Y -620.007,Z 446.260,A 0.000,B 0.000,C 90.000,E1 262.761} C_DIS
LIN {X 0.261,Y -615.694,Z 446.251,A 0.000,B 0.000,C 90.000,E1 261.197} C_DIS
LIN {X -0.207,Y -611.139,Z 446.243,A 0.000,B 0.000,C 90.000,E1 259.690} C_DIS
LIN {X 0.318,Y -607.234,Z 446.235,A 0.000,B 0.000,C 90.000,E1 258.342} C_DIS
LIN {X -0.266,Y -604.039,Z 446.230,A 0.000,B 0.000,C 90.000,E1 257.353} C_DIS
LIN {X 0.270,Y -599.968,Z 446.222,A 0.000,B 0.000,C 90.000,E1 255.992} C_DIS
LIN {X -0.281,Y -596.588,Z 446.217,A 0.000,B 0.000,C 90.000,E1 254.991} C_DIS
LIN {X -0.018,Y -591.434,Z 446.208,A 0.000,B 0.000,C 90.000,E1 253.378} C_DIS
LIN {X 0.036,Y -587.907,Z 446.202,A 0.000,B 0.000,C 90.000,E1 252.308} C_DIS
LIN {X 0.070,Y -583.426,Z 446.194,A 0.000,B 0.000,C 90.000,E1 250.967} C_DIS
LIN {X 0.222,Y -577.891,Z 446.185,A 0.000,B 0.000,C 90.000,E1 249.337} C_DIS
LIN {X -0.082,Y -574.029,Z 446.179,A 0.000,B 0.000,C 90.000,E1 248.284} C_DIS
LIN {X 0.095,Y -570.052,Z 446.173,A 0.000,B 0.000,C 90.000,E1 247.177} C_DIS
LIN {X -0.085,Y -565.962,Z 446.167,A 0.000,B 0.000,C 90.000,E1 246.102} C_DIS
LIN {X 0.004,Y -560.715,Z 446.160,A 0.000,B 0.000,C 90.000,E1 244.717} C_DIS
LIN {X -0.297,Y -556.455,Z 446.153,A 0.000,B 0.000,C 90.000,E1 243.640} C_DIS
LIN {X -0.110,Y -550.001,Z 446.144,A 0.000,B 0.000,C 90.000,E1 241.948} C_DIS
LIN {X 0.158,Y -542.650,Z 446.133,A 0.000,B 0.000,C 90.000,E1 239.950} C_DIS
LIN {X -0.165,Y -535.456,Z 446.122,A 0.000,B 0.000,C 90.000,E1 237.995} C_DIS
LIN {X -0.348,Y -529.218,Z 446.113,A 0.000,B 0.000,C 90.000,E1 236.294} C_DIS
LIN {X 0.314,Y -521.982,Z 446.101,A 0.000,B 0.000,C 90.000,E1 234.196} C_DIS
LIN {X -0.055,Y -514.832,Z 446.090,A 0.000,B 0.000,C 90.000,E1 232.190} C_DIS
LIN {X 0.073,Y -505.563,Z 446.074,A 0.000,B 0.000,C 90.000,E1 229.218} C_DIS
LIN {X 0.165,Y -501.138,Z 446.065,A 0.000,B 0.000,C 90.000,E1 227.715} C_DIS
LIN {X 0.138,Y -496.809,Z 446.057,A 0.000,B 0.000,C 90.000,E1 226.215} C_DIS
LIN {X -0.141,Y -491.704,Z 446.047,A 0.000,B 0.000,C 90.000,E1 224.433} C_DIS
LIN {X -0.179,Y -486.783,Z 446.037,A 0.000,B 0.000,C 90.000,E1 222.609} C_DIS
LIN {X -0.167,Y -481.224,Z 446.025,A 0.000,B 0.000,C 90.000,E1 220.458} C_DIS
LIN {X 0.123,Y -475.884,Z 446.013,A 0.000,B 0.000,C 90.000,E1 218.257} C_DIS
LIN {X -0.036,Y -468.744,Z 445.995,A 0.000,B 0.000,C 90.000,E1 215.152} C_DIS
LIN {X 0.098,Y -464.676,Z 445.985,A 0.000,B 0.000,C 90.000,E1 213.245} C_DIS
LIN {X 0.004,Y -459.412,Z 445.971,A 0.000,B 0.000,C 90.000,E1 210.718} C_DIS
LIN {X -0.151,Y -455.534,Z 445.960,A 0.000,B 0.000,C 90.000,E1 208.821} C_DIS
LIN {X -0.079,Y -452.275,Z 445.951,A 0.000,B 0.000,C 90.000,E1 207.206} C_DIS
LIN {X 0.048,Y -449.628,Z 445.944,A 0.000,B 0.000,C 90.000,E1 205.899} C_DIS
LIN {X -0.066,Y -444.904,Z 445.931,A 0.000,B 0.000,C 90.000,E1 203.643} C_DIS
LIN {X -0.179,Y -441.587,Z 445.922,A 0.000,B 0.000,C 90.000,E1 202.025} C_DIS
LIN {X -0.013,Y -437.069,Z 445.910,A 0.000,B 0.000,C 90.000,E1 199.704} C_DIS
LIN {X 0.116,Y -432.337,Z 445.895,A 0.000,B 0.000,C 90.000,E1 197.040} C_DIS
LIN {X -0.056,Y -429.047,Z 445.884,A 0.000,B 0.000,C 90.000,E1 195.064} C_DIS
LIN {X -0.020,Y -425.475,Z 445.871,A 0.000,B 0.000,C 90.000,E1 192.715} C_DIS
LIN {X 0.075,Y -421.305,Z 445.854,A 0.000,B 0.000,C 90.000,E1 189.670} C_DIS
LIN {X 0.085,Y -418.427,Z 445.841,A 0.000,B 0.000,C 90.000,E1 187.296} C_DIS
LIN {X -0.079,Y -415.867,Z 445.827,A 0.000,B 0.000,C 90.000,E1 184.935} C_DIS
LIN {X 0.075,Y -413.255,Z 445.812,A 0.000,B 0.000,C 90.000,E1 182.178} C_DIS
LIN {X 0.103,Y -410.655,Z 445.791,A 0.000,B 0.000,C 90.000,E1 178.396} C_DIS
LIN {X 0.076,Y -409.285,Z 445.770,A 0.000,B 0.000,C 90.000,E1 174.609} C_DIS
LIN {X -0.188,Y -409.338,Z 445.749,A 0.000,B 0.000,C 90.000,E1 170.849} C_DIS
LIN {X -0.142,Y -410.521,Z 445.728,A 0.000,B 0.000,C 90.000,E1 167.048} C_DIS
LIN {X 0.077,Y -412.281,Z 445.711,A 0.000,B 0.000,C 90.000,E1 163.921} C_DIS
LIN {X -0.202,Y -415.532,Z 445.690,A 0.000,B 0.000,C 90.000,E1 160.188} C_DIS
LIN {X 0.148,Y -418.540,Z 445.675,A 0.000,B 0.000,C 90.000,E1 157.411} C_DIS
LIN {X 0.043,Y -421.629,Z 445.661,A 0.000,B 0.000,C 90.000,E1 155.049} C_DIS
LIN {X -0.040,Y -425.447,Z 445.646,A 0.000,B 0.000,C 90.000,E1 152.359} C_DIS
LIN {X 0.048,Y -428.091,Z 445.637,A 0.000,B 0.000,C 90.000,E1 150.667} C_DIS
LIN {X 0.030,Y -430.805,Z 445.628,A 0.000,B 0.000,C 90.000,E1 148.997} C_DIS
LIN {X 0.003,Y -436.004,Z 445.611,A 0.000,B 0.000,C 90.000,E1 146.008} C_DIS
LIN {X -0.067,Y -439.706,Z 445.600,A 0.000,B 0.000,C 90.000,E1 144.036} C_DIS
LIN {X -0.064,Y -445.039,Z 445.586,A 0.000,B 0.000,C 90.000,E1 141.412} C_DIS
LIN {X -0.092,Y -449.885,Z 445.573,A 0.000,B 0.000,C 90.000,E1 139.138} C_DIS
LIN {X -0.040,Y -453.329,Z 445.564,A 0.000,B 0.000,C 90.000,E1 137.514} C_DIS
LIN {X 0.077,Y -456.628,Z 445.555,A 0.000,B 0.000,C 90.000,E1 135.891} C_DIS
LIN {X 0.168,Y -458.377,Z 445.550,A 0.000,B 0.000,C 90.000,E1 134.919} C_DIS
LIN {X 0.280,Y -460.014,Z 445.544,A 0.000,B 0.000,C 90.000,E1 133.947} C_DIS
LIN {X 0.092,Y -461.345,Z 445.539,A 0.000,B 0.000,C 90.000,E1 133.014} C_DIS
LIN {X 0.184,Y -462.162,Z 445.536,A 0.000,B 0.000,C 90.000,E1 132.366} C_DIS
LIN {X -0.240,Y -463.320,Z 445.528,A 0.000,B 0.000,C 90.000,E1 131.148} C_DIS
LIN {X -0.044,Y -463.832,Z 445.523,A 0.000,B 0.000,C 90.000,E1 130.172} C_DIS
LIN {X 0.159,Y -463.857,Z 445.518,A 0.000,B 0.000,C 90.000,E1 129.197} C_DIS
LIN {X -0.088,Y -463.765,Z 445.516,A 0.000,B 0.000,C 90.000,E1 128.910} C_DIS
LIN {X 0.109,Y -463.089,Z 445.511,A 0.000,B 0.000,C 90.000,E1 127.935} C_DIS
LIN {X 0.007,Y -462.056,Z 445.506,A 0.000,B 0.000,C 90.000,E1 126.996} C_DIS
LIN {X -0.124,Y -461.223,Z 445.502,A 0.000,B 0.000,C 90.000,E1 126.377} C_DIS
LIN {X 0.129,Y -459.654,Z 445.497,A 0.000,B 0.000,C 90.000,E1 125.391} C_DIS
LIN {X -0.016,Y -457.608,Z 445.491,A 0.000,B 0.000,C 90.000,E1 124.452} C_DIS
LIN {X 0.204,Y -456.137,Z 445.488,A 0.000,B 0.000,C 90.000,E1 123.785} C_DIS
LIN {X -0.143,Y -452.637,Z 445.481,A 0.000,B 0.000,C 90.000,E1 122.546} C_DIS
LIN {X -0.162,Y -448.836,Z 445.474,A 0.000,B 0.000,C 90.000,E1 121.258} C_DIS
LIN {X 0.068,Y -445.793,Z 445.468,A 0.000,B 0.000,C 90.000,E1 120.256} C_DIS
LIN {X 0.146,Y -440.478,Z 445.459,A 0.000,B 0.000,C 90.000,E1 118.615} C_DIS
LIN {X 0.059,Y -437.109,Z 445.454,A 0.000,B 0.000,C 90.000,E1 117.641} C_DIS
LIN {X 0.019,Y -437.098,Z 445.454,A 0.000,B 0.000,C 90.000,E1 117.641} C_DIS
LIN {X -0.069,Y -444.519,Z 445.439,A 0.000,B 0.000,C 90.000,E1 115.027} C_DIS
LIN {X 0.099,Y -446.664,Z 445.434,A 0.000,B 0.000,C 90.000,E1 114.027} C_DIS
LIN {X -0.035,Y -455.388,Z 445.414,A 0.000,B 0.000,C 90.000,E1 110.482} C_DIS
LIN {X 0.190,Y -457.187,Z 445.410,A 0.000,B 0.000,C 90.000,E1 109.812} C_DIS
LIN {X 0.058,Y -466.580,Z 445.385,A 0.000,B 0.000,C 90.000,E1 105.371} C_DIS
LIN {X -0.019,Y -467.368,Z 445.384,A 0.000,B 0.000,C 90.000,E1 105.064} C_DIS
LIN {X -0.217,Y -468.017,Z 445.382,A 0.000,B 0.000,C 90.000,E1 104.773} C_DIS
LIN {X 0.215,Y -476.230,Z 445.356,A 0.000,B 0.000,C 90.000,E1 100.018} C_DIS
LIN {X 0.000,Y -482.126,Z 445.330,A 0.000,B 0.000,C 90.000,E1 95.391} C_DIS
LIN {X -0.136,Y -484.085,Z 445.313,A 0.000,B 0.000,C 90.000,E1 92.293} C_DIS
LIN {X -0.197,Y -574.097,Z 445.313,A 0.000,B 0.000,C 90.000,E1 92.293} C_DIS
LIN {X 0.276,Y -576.734,Z 445.313,A 0.000,B 0.000,C 90.000,E1 92.236} C_DIS
LIN {X 0.018,Y -580.102,Z 445.312,A 0.000,B 0.000,C 90.000,E1 92.236} C_DIS
LIN {X -0.046,Y -585.569,Z 445.311,A 0.000,B 0.000,C 90.000,E1 92.007} C_DIS
LIN {X 0.238,Y -587.505,Z 445.310,A 0.000,B 0.000,C 90.000,E1 91.835} C_DIS
LIN {X 0.066,Y -592.189,Z 445.308,A 0.000,B 0.000,C 90.000,E1 91.375} C_DIS
LIN {X -0.209,Y -593.505,Z 445.306,A 0.000,B 0.000,C 90.000,E1 91.146} C_DIS
LIN {X 0.006,Y -594.560,Z 445.305,A 0.000,B 0.000,C 90.000,E1 90.859} C_DIS
LIN {X 0.225,Y -595.338,Z 445.303,A 0.000,B 0.000,C 90.000,E1 90.573} C_DIS
LIN {X -0.147,Y -595.524,Z 445.302,A 0.000,B 0.000,C 90.000,E1 90.344} C_DIS
LIN {X 0.079,Y -595.500,Z 445.300,A 0.000,B 0.000,C 90.000,E1 90.057} C_DIS
LIN {X -0.289,Y -594.666,Z 445.299,A 0.000,B 0.000,C 90.000,E1 89.828} C_DIS
LIN {X -0.062,Y -594.116,Z 445.297,A 0.000,B 0.000,C 90.000,E1 89.542} C_DIS
LIN {X 0.161,Y -593.034,Z 445.296,A 0.000,B 0.000,C 90.000,E1 89.255} C_DIS
LIN {X -0.025,Y -592.264,Z 445.295,A 0.000,B 0.000,C 90.000,E1 89.141} C_DIS
LIN {X 0.191,Y -590.335,Z 445.294,A 0.000,B 0.000,C 90.000,E1 88.854} C_DIS
LIN {X 0.002,Y -589.059,Z 445.293,A 0.000,B 0.000,C 90.000,E1 88.740} C_DIS
LIN {X 0.250,Y -586.012,Z 445.292,A 0.000,B 0.000,C 90.000,E1 88.453} C_DIS
LIN {X -0.223,Y -580.702,Z 445.290,A 0.000,B 0.000,C 90.000,E1 88.165} C_DIS
LIN {X 0.191,Y -575.563,Z 445.289,A 0.000,B 0.000,C 90.000,E1 87.993} C_DIS
LIN {X -0.266,Y -573.356,Z 445.289,A 0.000,B 0.000,C 90.000,E1 87.993} C_DIS
LIN {X 0.220,Y -485.813,Z 445.289,A 0.000,B 0.000,C 90.000,E1 87.936} C_DIS
LIN {X -0.088,Y -486.312,Z 445.282,A 0.000,B 0.000,C 90.000,E1 86.731} C_DIS
LIN {X 0.047,Y -486.315,Z 445.278,A 0.000,B 0.000,C 90.000,E1 86.102} C_DIS
LIN {X 0.120,Y -484.616,Z 445.253,A 0.000,B 0.000,C 90.000,E1 81.489} C_DIS
LIN {X -0.001,Y -480.547,Z 445.227,A 0.000,B 0.000,C 90.000,E1 76.881} C_DIS
LIN {X -0.089,Y -474.300,Z 445.201,A 0.000,B 0.000,C 90.000,E1 72.236} C_DIS
LIN {X -0.268,Y -473.879,Z 445.200,A 0.000,B 0.000,C 90.000,E1 71.945} C_DIS
LIN {X -0.141,Y -466.276,Z 445.175,A 0.000,B 0.000,C 90.000,E1 67.539} C_DIS
LIN {X -0.198,Y -465.846,Z 445.173,A 0.000,B 0.000,C 90.000,E1 67.230} C_DIS
LIN {X -0.256,Y -465.269,Z 445.172,A 0.000,B 0.000,C 90.000,E1 66.922} C_DIS
LIN {X 0.060,Y -461.742,Z 445.163,A 0.000,B 0.000,C 90.000,E1 65.305} C_DIS
LIN {X 0.020,Y -461.744,Z 445.163,A 0.000,B 0.000,C 90.000,E1 65.305} C_DIS
LIN {X -0.006,Y -474.245,Z 445.153,A 0.000,B 0.000,C 90.000,E1 63.563} C_DIS
LIN {X -0.119,Y -481.861,Z 445.147,A 0.000,B 0.000,C 90.000,E1 62.487} C_DIS
LIN {X 0.091,Y -487.112,Z 445.143,A 0.000,B 0.000,C 90.000,E1 61.691} C_DIS
LIN {X 0.120,Y -491.838,Z 445.139,A 0.000,B 0.000,C 90.000,E1 60.923} C_DIS
LIN {X -0.038,Y -495.387,Z 445.135,A 0.000,B 0.000,C 90.000,E1 60.333} C_DIS
LIN {X -0.173,Y -498.578,Z 445.132,A 0.000,B 0.000,C 90.000,E1 59.744} C_DIS
LIN {X -0.227,Y -502.061,Z 445.128,A 0.000,B 0.000,C 90.000,E1 58.997} C_DIS
LIN {X -0.122,Y -503.941,Z 445.125,A 0.000,B 0.000,C 90.000,E1 58.535} C_DIS
LIN {X 0.066,Y -506.113,Z 445.122,A 0.000,B 0.000,C 90.000,E1 57.916} C_DIS
LIN {X -0.318,Y -507.107,Z 445.120,A 0.000,B 0.000,C 90.000,E1 57.661} C_DIS
LIN {X -0.106,Y -508.751,Z 445.117,A 0.000,B 0.000,C 90.000,E1 57.041} C_DIS
LIN {X 0.030,Y -510.793,Z 445.112,A 0.000,B 0.000,C 90.000,E1 56.135} C_DIS
LIN {X -0.013,Y -511.796,Z 445.109,A 0.000,B 0.000,C 90.000,E1 55.548} C_DIS
LIN {X -0.266,Y -512.850,Z 445.104,A 0.000,B 0.000,C 90.000,E1 54.689} C_DIS
LIN {X -0.086,Y -513.477,Z 445.099,A 0.000,B 0.000,C 90.000,E1 53.783} C_DIS
LIN {X 0.252,Y -513.671,Z 445.091,A 0.000,B 0.000,C 90.000,E1 52.271} C_DIS
LIN {X 0.099,Y -513.605,Z 445.087,A 0.000,B 0.000,C 90.000,E1 51.698} C_DIS
LIN {X 0.189,Y -513.313,Z 445.082,A 0.000,B 0.000,C 90.000,E1 50.803} C_DIS
LIN {X 0.279,Y -512.866,Z 445.077,A 0.000,B 0.000,C 90.000,E1 49.908} C_DIS
LIN {X -0.199,Y -511.746,Z 445.069,A 0.000,B 0.000,C 90.000,E1 48.485} C_DIS
LIN {X -0.016,Y -510.467,Z 445.061,A 0.000,B 0.000,C 90.000,E1 46.986} C_DIS
LIN {X -0.099,Y -509.340,Z 445.055,A 0.000,B 0.000,C 90.000,E1 45.810} C_DIS
LIN {X 0.041,Y -507.026,Z 445.041,A 0.000,B 0.000,C 90.000,E1 43.419} C_DIS
LIN {X -0.127,Y -505.038,Z 445.030,A 0.000,B 0.000,C 90.000,E1 41.353} C_DIS
LIN {X -0.034,Y -503.579,Z 445.021,A 0.000,B 0.000,C 90.000,E1 39.850} C_DIS
LIN {X -0.007,Y -501.850,Z 445.011,A 0.000,B 0.000,C 90.000,E1 38.051} C_DIS
LIN {X -0.287,Y -500.325,Z 445.003,A 0.000,B 0.000,C 90.000,E1 36.583} C_DIS
LIN {X -0.083,Y -498.944,Z 444.996,A 0.000,B 0.000,C 90.000,E1 35.358} C_DIS
LIN {X 0.083,Y -497.221,Z 444.988,A 0.000,B 0.000,C 90.000,E1 33.833} C_DIS
LIN {X 0.088,Y -495.754,Z 444.981,A 0.000,B 0.000,C 90.000,E1 32.625} C_DIS
LIN {X 0.192,Y -493.400,Z 444.971,A 0.000,B 0.000,C 90.000,E1 30.797} C_DIS
LIN {X -0.018,Y -491.012,Z 444.961,A 0.000,B 0.000,C 90.000,E1 28.999} C_DIS
LIN {X -0.080,Y -488.297,Z 444.949,A 0.000,B 0.000,C 90.000,E1 26.873} C_DIS
LIN {X 0.003,Y -486.220,Z 444.939,A 0.000,B 0.000,C 90.000,E1 25.027} C_DIS
LIN {X -0.134,Y -483.584,Z 444.924,A 0.000,B 0.000,C 90.000,E1 22.280} C_DIS
LIN {X -0.098,Y -481.790,Z 444.910,A 0.000,B 0.000,C 90.000,E1 19.812} C_DIS
LIN {X 0.021,Y -480.649,Z 444.900,A 0.000,B 0.000,C 90.000,E1 17.946} C_DIS
LIN {X -0.042,Y -479.164,Z 444.888,A 0.000,B 0.000,C 90.000,E1 15.788} C_DIS
LIN {X -0.130,Y -477.884,Z 444.877,A 0.000,B 0.000,C 90.000,E1 13.939} C_DIS
LIN {X -0.016,Y -476.461,Z 444.862,A 0.000,B 0.000,C 90.000,E1 11.130} C_DIS
LIN {X 0.124,Y -475.656,Z 444.848,A 0.000,B 0.000,C 90.000,E1 8.624} C_DIS
LIN {X 0.031,Y -475.348,Z 444.834,A 0.000,B 0.000,C 90.000,E1 6.144} C_DIS
LIN {X -0.193,Y -475.520,Z 444.824,A 0.000,B 0.000,C 90.000,E1 4.302} C_DIS
LIN {X 0.235,Y -476.951,Z 444.803,A 0.000,B 0.000,C 90.000,E1 0.516} C_DIS
LIN {X -0.167,Y -479.721,Z 444.783,A 0.000,B 0.000,C 90.000,E1 357.020} C_DIS
LIN {X -0.006,Y -482.216,Z 444.771,A 0.000,B 0.000,C 90.000,E1 354.837} C_DIS
LIN {X 0.138,Y -485.506,Z 444.758,A 0.000,B 0.000,C 90.000,E1 352.356} C_DIS
LIN {X -0.037,Y -489.296,Z 444.744,A 0.000,B 0.000,C 90.000,E1 349.926} C_DIS
LIN {X -0.202,Y -496.602,Z 444.722,A 0.000,B 0.000,C 90.000,E1 345.992} C_DIS
LIN {X -0.023,Y -503.488,Z 444.705,A 0.000,B 0.000,C 90.000,E1 342.960} C_DIS
LIN {X -0.263,Y -511.075,Z 444.689,A 0.000,B 0.000,C 90.000,E1 340.007} C_DIS
LIN {X 0.315,Y -515.022,Z 444.681,A 0.000,B 0.000,C 90.000,E1 338.465} C_DIS
LIN {X -0.180,Y -519.018,Z 444.672,A 0.000,B 0.000,C 90.000,E1 337.050} C_DIS
LIN {X 0.283,Y -522.997,Z 444.664,A 0.000,B 0.000,C 90.000,E1 335.537} C_DIS
LIN {X 0.213,Y -528.571,Z 444.653,A 0.000,B 0.000,C 90.000,E1 333.512} C_DIS
LIN {X -0.140,Y -533.335,Z 444.643,A 0.000,B 0.000,C 90.000,E1 331.820} C_DIS
LIN {X 0.192,Y -535.772,Z 444.639,A 0.000,B 0.000,C 90.000,E1 330.923} C_DIS
LIN {X 0.254,Y -540.658,Z 444.629,A 0.000,B 0.000,C 90.000,E1 329.203} C_DIS
LIN {X -0.049,Y -545.522,Z 444.620,A 0.000,B 0.000,C 90.000,E1 327.533} C_DIS
LIN {X 0.081,Y -551.035,Z 444.609,A 0.000,B 0.000,C 90.000,E1 325.548} C_DIS
LIN {X -0.239,Y -556.649,Z 444.598,A 0.000,B 0.000,C 90.000,E1 323.623} C_DIS
LIN {X -0.071,Y -562.406,Z 444.587,A 0.000,B 0.000,C 90.000,E1 321.662} C_DIS
LIN {X 0.036,Y -570.171,Z 444.573,A 0.000,B 0.000,C 90.000,E1 319.175} C_DIS
LIN {X 0.051,Y -573.639,Z 444.567,A 0.000,B 0.000,C 90.000,E1 318.081} C_DIS
LIN {X -0.023,Y -578.650,Z 444.558,A 0.000,B 0.000,C 90.000,E1 316.458} C_DIS
LIN {X -0.277,Y -584.522,Z 444.548,A 0.000,B 0.000,C 90.000,E1 314.595} C_DIS
LIN {X -0.017,Y -592.174,Z 444.534,A 0.000,B 0.000,C 90.000,E1 312.162} C_DIS
LIN {X 0.083,Y -596.338,Z 444.527,A 0.000,B 0.000,C 90.000,E1 310.825} C_DIS
LIN {X -0.073,Y -600.373,Z 444.520,A 0.000,B 0.000,C 90.000,E1 309.519} C_DIS
LIN {X 0.232,Y -604.347,Z 444.512,A 0.000,B 0.000,C 90.000,E1 308.177} C_DIS
LIN {X 0.224,Y -608.183,Z 444.505,A 0.000,B 0.000,C 90.000,E1 306.870} C_DIS
LIN {X 0.202,Y -612.664,Z 444.496,A 0.000,B 0.000,C 90.000,E1 305.311} C_DIS
LIN {X 0.172,Y -615.464,Z 444.491,A 0.000,B 0.000,C 90.000,E1 304.278} C_DIS
LIN {X 0.183,Y -618.206,Z 444.485,A 0.000,B 0.000,C 90.000,E1 303.245} C_DIS
LIN {X -0.003,Y -622.159,Z 444.476,A 0.000,B 0.000,C 90.000,E1 301.720} C_DIS
LIN {X 0.293,Y -624.680,Z 444.471,A 0.000,B 0.000,C 90.000,E1 300.669} C_DIS
LIN {X 0.102,Y -627.646,Z 444.464,A 0.000,B 0.000,C 90.000,E1 299.411} C_DIS
LIN {X -0.022,Y -631.057,Z 444.455,A 0.000,B 0.000,C 90.000,E1 297.897} C_DIS
LIN {X 0.145,Y -633.855,Z 444.448,A 0.000,B 0.000,C 90.000,E1 296.616} C_DIS
LIN {X 0.358,Y -636.490,Z 444.441,A 0.000,B 0.000,C 90.000,E1 295.335} C_DIS
LIN {X 0.238,Y -637.939,Z 444.437,A 0.000,B 0.000,C 90.000,E1 294.591} C_DIS
LIN {X 0.252,Y -640.243,Z 444.430,A 0.000,B 0.000,C 90.000,E1 293.334} C_DIS
LIN {X 0.172,Y -643.109,Z 444.420,A 0.000,B 0.000,C 90.000,E1 291.589} C_DIS
LIN {X -0.095,Y -645.706,Z 444.410,A 0.000,B 0.000,C 90.000,E1 289.866} C_DIS
LIN {X 0.166,Y -647.337,Z 444.403,A 0.000,B 0.000,C 90.000,E1 288.598} C_DIS
LIN {X -0.356,Y -648.675,Z 444.397,A 0.000,B 0.000,C 90.000,E1 287.402} C_DIS
LIN {X -0.046,Y -649.855,Z 444.390,A 0.000,B 0.000,C 90.000,E1 286.134} C_DIS
LIN {X -0.075,Y -650.946,Z 444.383,A 0.000,B 0.000,C 90.000,E1 284.898} C_DIS
LIN {X -0.166,Y -651.286,Z 444.380,A 0.000,B 0.000,C 90.000,E1 284.411} C_DIS
LIN {X 0.338,Y -651.983,Z 444.372,A 0.000,B 0.000,C 90.000,E1 282.883} C_DIS
LIN {X -0.302,Y -652.375,Z 444.366,A 0.000,B 0.000,C 90.000,E1 281.951} C_DIS
LIN {X 0.101,Y -652.648,Z 444.358,A 0.000,B 0.000,C 90.000,E1 280.433} C_DIS
LIN {X -0.285,Y -652.581,Z 444.354,A 0.000,B 0.000,C 90.000,E1 279.726} C_DIS
LIN {X 0.266,Y -652.335,Z 444.348,A 0.000,B 0.000,C 90.000,E1 278.690} C_DIS
LIN {X -0.096,Y -651.579,Z 444.340,A 0.000,B 0.000,C 90.000,E1 277.239} C_DIS
LIN {X -0.192,Y -650.833,Z 444.335,A 0.000,B 0.000,C 90.000,E1 276.258} C_DIS
LIN {X -0.141,Y -650.103,Z 444.331,A 0.000,B 0.000,C 90.000,E1 275.511} C_DIS
LIN {X 0.165,Y -648.524,Z 444.324,A 0.000,B 0.000,C 90.000,E1 274.245} C_DIS
LIN {X -0.213,Y -646.513,Z 444.317,A 0.000,B 0.000,C 90.000,E1 273.037} C_DIS
LIN {X -0.023,Y -644.278,Z 444.310,A 0.000,B 0.000,C 90.000,E1 271.776} C_DIS
LIN {X -0.297,Y -642.260,Z 444.304,A 0.000,B 0.000,C 90.000,E1 270.802} C_DIS
LIN {X 0.211,Y -638.969,Z 444.296,A 0.000,B 0.000,C 90.000,E1 269.255} C_DIS
LIN {X 0.275,Y -635.848,Z 444.289,A 0.000,B 0.000,C 90.000,E1 267.993} C_DIS
LIN {X 0.029,Y -631.852,Z 444.281,A 0.000,B 0.000,C 90.000,E1 266.502} C_DIS
LIN {X -0.031,Y -628.496,Z 444.274,A 0.000,B 0.000,C 90.000,E1 265.241} C_DIS
LIN {X 0.287,Y -624.362,Z 444.265,A 0.000,B 0.000,C 90.000,E1 263.685} C_DIS
LIN {X -0.163,Y -621.515,Z 444.259,A 0.000,B 0.000,C 90.000,E1 262.704} C_DIS
LIN {X 0.097,Y -617.161,Z 444.251,A 0.000,B 0.000,C 90.000,E1 261.141} C_DIS
LIN {X 0.009,Y -613.367,Z 444.244,A 0.000,B 0.000,C 90.000,E1 259.859} C_DIS
LIN {X 0.204,Y -608.656,Z 444.235,A 0.000,B 0.000,C 90.000,E1 258.285} C_DIS
LIN {X -0.232,Y -605.424,Z 444.229,A 0.000,B 0.000,C 90.000,E1 257.285} C_DIS
LIN {X 0.194,Y -601.337,Z 444.222,A 0.000,B 0.000,C 90.000,E1 255.936} C_DIS
LIN {X 0.106,Y -597.037,Z 444.215,A 0.000,B 0.000,C 90.000,E1 254.629} C_DIS
LIN {X 0.207,Y -591.859,Z 444.206,A 0.000,B 0.000,C 90.000,E1 253.032} C_DIS
LIN {X -0.349,Y -585.560,Z 444.196,A 0.000,B 0.000,C 90.000,E1 251.221} C_DIS
LIN {X 0.195,Y -580.892,Z 444.188,A 0.000,B 0.000,C 90.000,E1 249.826} C_DIS
LIN {X 0.084,Y -578.092,Z 444.184,A 0.000,B 0.000,C 90.000,E1 249.028} C_DIS
LIN {X -0.215,Y -574.167,Z 444.178,A 0.000,B 0.000,C 90.000,E1 247.975} C_DIS
LIN {X -0.208,Y -569.103,Z 444.170,A 0.000,B 0.000,C 90.000,E1 246.613} C_DIS
LIN {X -0.254,Y -562.813,Z 444.161,A 0.000,B 0.000,C 90.000,E1 244.973} C_DIS
LIN {X -0.024,Y -558.570,Z 444.155,A 0.000,B 0.000,C 90.000,E1 243.845} C_DIS
LIN {X 0.198,Y -552.095,Z 444.145,A 0.000,B 0.000,C 90.000,E1 242.153} C_DIS
LIN {X 0.058,Y -543.638,Z 444.133,A 0.000,B 0.000,C 90.000,E1 239.921} C_DIS
LIN {X 0.227,Y -537.461,Z 444.124,A 0.000,B 0.000,C 90.000,E1 238.201} C_DIS
LIN {X 0.093,Y -532.267,Z 444.116,A 0.000,B 0.000,C 90.000,E1 236.786} C_DIS
LIN {X -0.261,Y -528.092,Z 444.109,A 0.000,B 0.000,C 90.000,E1 235.674} C_DIS
LIN {X -0.012,Y -521.900,Z 444.100,A 0.000,B 0.000,C 90.000,E1 233.909} C_DIS
LIN {X 0.275,Y -513.877,Z 444.087,A 0.000,B 0.000,C 90.000,E1 231.537} C_DIS
LIN {X -0.250,Y -505.650,Z 444.072,A 0.000,B 0.000,C 90.000,E1 228.933} C_DIS
LIN {X -0.107,Y -499.519,Z 444.060,A 0.000,B 0.000,C 90.000,E1 226.824} C_DIS
LIN {X 0.217,Y -493.542,Z 444.048,A 0.000,B 0.000,C 90.000,E1 224.676} C_DIS
LIN {X -0.313,Y -487.732,Z 444.037,A 0.000,B 0.000,C 90.000,E1 222.609} C_DIS
LIN {X 0.093,Y -482.179,Z 444.025,A 0.000,B 0.000,C 90.000,E1 220.415} C_DIS
LIN {X 0.042,Y -476.823,Z 444.013,A 0.000,B 0.000,C 90.000,E1 218.257} C_DIS
LIN {X 0.078,Y -468.939,Z 443.994,A 0.000,B 0.000,C 90.000,E1 214.818} C_DIS
LIN {X 0.072,Y -465.530,Z 443.985,A 0.000,B 0.000,C 90.000,E1 213.245} C_DIS
LIN {X 0.005,Y -460.240,Z 443.971,A 0.000,B 0.000,C 90.000,E1 210.718} C_DIS
LIN {X -0.131,Y -456.340,Z 443.960,A 0.000,B 0.000,C 90.000,E1 208.821} C_DIS
LIN {X -0.044,Y -453.053,Z 443.951,A 0.000,B 0.000,C 90.000,E1 207.206} C_DIS
LIN {X -0.026,Y -449.705,Z 443.942,A 0.000,B 0.000,C 90.000,E1 205.591} C_DIS
LIN {X -0.130,Y -444.968,Z 443.930,A 0.000,B 0.000,C 90.000,E1 203.334} C_DIS
LIN {X 0.024,Y -440.945,Z 443.919,A 0.000,B 0.000,C 90.000,E1 201.354} C_DIS
LIN {X -0.074,Y -437.132,Z 443.908,A 0.000,B 0.000,C 90.000,E1 199.396} C_DIS
LIN {X 0.049,Y -432.424,Z 443.893,A 0.000,B 0.000,C 90.000,E1 196.732} C_DIS
LIN {X 0.077,Y -429.659,Z 443.884,A 0.000,B 0.000,C 90.000,E1 195.064} C_DIS
LIN {X -0.058,Y -427.060,Z 443.875,A 0.000,B 0.000,C 90.000,E1 193.411} C_DIS
LIN {X -0.163,Y -423.647,Z 443.861,A 0.000,B 0.000,C 90.000,E1 191.074} C_DIS
LIN {X 0.063,Y -420.184,Z 443.846,A 0.000,B 0.000,C 90.000,E1 188.341} C_DIS
LIN {X -0.014,Y -417.806,Z 443.835,A 0.000,B 0.000,C 90.000,E1 186.315} C_DIS
LIN {X 0.164,Y -416.017,Z 443.826,A 0.000,B 0.000,C 90.000,E1 184.588} C_DIS
LIN {X -0.117,Y -413.504,Z 443.810,A 0.000,B 0.000,C 90.000,E1 181.892} C_DIS
LIN {X -0.071,Y -411.337,Z 443.793,A 0.000,B 0.000,C 90.000,E1 178.797} C_DIS
LIN {X -0.081,Y -410.141,Z 443.778,A 0.000,B 0.000,C 90.000,E1 176.045} C_DIS
LIN {X 0.064,Y -409.809,Z 443.751,A 0.000,B 0.000,C 90.000,E1 171.197} C_DIS
LIN {X 0.067,Y -411.011,Z 443.728,A 0.000,B 0.000,C 90.000,E1 167.061} C_DIS
LIN {X -0.132,Y -412.580,Z 443.713,A 0.000,B 0.000,C 90.000,E1 164.338} C_DIS
LIN {X -0.004,Y -415.729,Z 443.692,A 0.000,B 0.000,C 90.000,E1 160.550} C_DIS
LIN {X -0.099,Y -419.529,Z 443.673,A 0.000,B 0.000,C 90.000,E1 157.155} C_DIS
LIN {X 0.165,Y -423.123,Z 443.658,A 0.000,B 0.000,C 90.000,E1 154.409} C_DIS
LIN {X 0.105,Y -428.219,Z 443.639,A 0.000,B 0.000,C 90.000,E1 151.051} C_DIS
LIN {X -0.119,Y -432.030,Z 443.626,A 0.000,B 0.000,C 90.000,E1 148.742} C_DIS
LIN {X -0.135,Y -436.793,Z 443.612,A 0.000,B 0.000,C 90.000,E1 146.087} C_DIS
LIN {X -0.191,Y -440.567,Z 443.601,A 0.000,B 0.000,C 90.000,E1 144.116} C_DIS
LIN {X 0.113,Y -445.995,Z 443.586,A 0.000,B 0.000,C 90.000,E1 141.457} C_DIS
LIN {X -0.170,Y -450.984,Z 443.573,A 0.000,B 0.000,C 90.000,E1 139.218} C_DIS
LIN {X 0.239,Y -454.521,Z 443.564,A 0.000,B 0.000,C 90.000,E1 137.553} C_DIS
LIN {X 0.015,Y -457.305,Z 443.557,A 0.000,B 0.000,C 90.000,E1 136.296} C_DIS
LIN {X 0.151,Y -459.786,Z 443.550,A 0.000,B 0.000,C 90.000,E1 135.000} C_DIS
LIN {X 0.234,Y -460.982,Z 443.547,A 0.000,B 0.000,C 90.000,E1 134.352} C_DIS
LIN {X 0.057,Y -462.503,Z 443.541,A 0.000,B 0.000,C 90.000,E1 133.419} C_DIS
LIN {X -0.045,Y -464.181,Z 443.534,A 0.000,B 0.000,C 90.000,E1 132.162} C_DIS
LIN {X -0.186,Y -465.065,Z 443.529,A 0.000,B 0.000,C 90.000,E1 131.229} C_DIS
LIN {X 0.032,Y -465.642,Z 443.524,A 0.000,B 0.000,C 90.000,E1 130.253} C_DIS
LIN {X -0.156,Y -465.783,Z 443.520,A 0.000,B 0.000,C 90.000,E1 129.644} C_DIS
LIN {X 0.017,Y -465.728,Z 443.517,A 0.000,B 0.000,C 90.000,E1 128.991} C_DIS
LIN {X 0.239,Y -465.149,Z 443.511,A 0.000,B 0.000,C 90.000,E1 128.016} C_DIS
LIN {X 0.163,Y -464.189,Z 443.506,A 0.000,B 0.000,C 90.000,E1 127.076} C_DIS
LIN {X 0.075,Y -462.863,Z 443.501,A 0.000,B 0.000,C 90.000,E1 126.137} C_DIS
LIN {X -0.049,Y -461.824,Z 443.497,A 0.000,B 0.000,C 90.000,E1 125.518} C_DIS
LIN {X 0.209,Y -459.851,Z 443.492,A 0.000,B 0.000,C 90.000,E1 124.532} C_DIS
LIN {X 0.182,Y -457.564,Z 443.487,A 0.000,B 0.000,C 90.000,E1 123.579} C_DIS
LIN {X -0.144,Y -454.013,Z 443.480,A 0.000,B 0.000,C 90.000,E1 122.339} C_DIS
LIN {X -0.145,Y -450.103,Z 443.472,A 0.000,B 0.000,C 90.000,E1 121.052} C_DIS
LIN {X -0.124,Y -446.965,Z 443.467,A 0.000,B 0.000,C 90.000,E1 120.079} C_DIS
LIN {X 0.020,Y -444.825,Z 443.463,A 0.000,B 0.000,C 90.000,E1 119.411} C_DIS
LIN {X 0.037,Y -440.370,Z 443.456,A 0.000,B 0.000,C 90.000,E1 118.103} C_DIS
LIN {X -0.043,Y -437.820,Z 443.452,A 0.000,B 0.000,C 90.000,E1 117.385} C_DIS
LIN {X -0.083,Y -437.805,Z 443.452,A 0.000,B 0.000,C 90.000,E1 117.385} C_DIS
LIN {X -0.040,Y -444.118,Z 443.440,A 0.000,B 0.000,C 90.000,E1 115.155} C_DIS
LIN {X 0.000,Y -445.020,Z 443.438,A 0.000,B 0.000,C 90.000,E1 114.823} C_DIS
LIN {X 0.089,Y -454.164,Z 443.416,A 0.000,B 0.000,C 90.000,E1 110.918} C_DIS
LIN {X 0.206,Y -456.823,Z 443.411,A 0.000,B 0.000,C 90.000,E1 109.939} C_DIS
LIN {X 0.108,Y -457.567,Z 443.409,A 0.000,B 0.000,C 90.000,E1 109.631} C_DIS
LIN {X 0.195,Y -466.268,Z 443.386,A 0.000,B 0.000,C 90.000,E1 105.481} C_DIS
LIN {X -0.203,Y -467.821,Z 443.383,A 0.000,B 0.000,C 90.000,E1 104.898} C_DIS
LIN {X -0.232,Y -476.028,Z 443.357,A 0.000,B 0.000,C 90.000,E1 100.197} C_DIS
LIN {X 0.072,Y -477.353,Z 443.350,A 0.000,B 0.000,C 90.000,E1 98.916} C_DIS
LIN {X 0.041,Y -481.961,Z 443.331,A 0.000,B 0.000,C 90.000,E1 95.511} C_DIS
LIN {X 0.175,Y -482.351,Z 443.327,A 0.000,B 0.000,C 90.000,E1 94.878} C_DIS
LIN {X -0.173,Y -485.421,Z 443.305,A 0.000,B 0.000,C 90.000,E1 90.917} C_DIS
LIN {X -0.035,Y -485.506,Z 443.302,A 0.000,B 0.000,C 90.000,E1 90.286} C_DIS
LIN {X -0.140,Y -486.373,Z 443.281,A 0.000,B 0.000,C 90.000,E1 86.617} C_DIS
LIN {X 0.170,Y -486.366,Z 443.279,A 0.000,B 0.000,C 90.000,E1 86.274} C_DIS
LIN {X -0.001,Y -485.230,Z 443.268,A 0.000,B 0.000,C 90.000,E1 84.147} C_DIS
LIN {X 0.258,Y -484.691,Z 443.254,A 0.000,B 0.000,C 90.000,E1 81.659} C_DIS
LIN {X 0.056,Y -484.471,Z 443.252,A 0.000,B 0.000,C 90.000,E1 81.376} C_DIS
LIN {X 0.059,Y -480.654,Z 443.228,A 0.000,B 0.000,C 90.000,E1 77.061} C_DIS
LIN {X 0.026,Y -480.391,Z 443.227,A 0.000,B 0.000,C 90.000,E1 76.756} C_DIS
LIN {X -0.201,Y -474.179,Z 443.201,A 0.000,B 0.000,C 90.000,E1 72.127} C_DIS
LIN {X 0.147,Y -472.367,Z 443.195,A 0.000,B 0.000,C 90.000,E1 71.148} C_DIS
LIN {X -0.168,Y -465.678,Z 443.173,A 0.000,B 0.000,C 90.000,E1 67.102} C_DIS
LIN {X -0.060,Y -462.203,Z 443.164,A 0.000,B 0.000,C 90.000,E1 65.537} C_DIS
LIN {X -0.100,Y -462.199,Z 443.164,A 0.000,B 0.000,C 90.000,E1 65.537} C_DIS
LIN {X 0.201,Y -473.787,Z 443.155,A 0.000,B 0.000,C 90.000,E1 63.896} C_DIS
LIN {X 0.087,Y -481.552,Z 443.149,A 0.000,B 0.000,C 90.000,E1 62.820} C_DIS
LIN {X 0.074,Y -487.882,Z 443.144,A 0.000,B 0.000,C 90.000,E1 61.897} C_DIS
LIN {X 0.109,Y -492.673,Z 443.140,A 0.000,B 0.000,C 90.000,E1 61.129} C_DIS
LIN {X -0.002,Y -497.101,Z 443.135,A 0.000,B 0.000,C 90.000,E1 60.383} C_DIS
LIN {X -0.121,Y -500.258,Z 443.132,A 0.000,B 0.000,C 90.000,E1 59.793} C_DIS
LIN {X -0.220,Y -503.088,Z 443.129,A 0.000,B 0.000,C 90.000,E1 59.203} C_DIS
LIN {X 0.200,Y -506.157,Z 443.125,A 0.000,B 0.000,C 90.000,E1 58.408} C_DIS
LIN {X -0.294,Y -508.278,Z 443.121,A 0.000,B 0.000,C 90.000,E1 57.867} C_DIS
LIN {X -0.170,Y -510.714,Z 443.116,A 0.000,B 0.000,C 90.000,E1 56.962} C_DIS
LIN {X 0.076,Y -512.096,Z 443.113,A 0.000,B 0.000,C 90.000,E1 56.342} C_DIS
LIN {X -0.038,Y -513.575,Z 443.108,A 0.000,B 0.000,C 90.000,E1 55.468} C_DIS
LIN {X 0.150,Y -514.498,Z 443.103,A 0.000,B 0.000,C 90.000,E1 54.562} C_DIS
LIN {X 0.002,Y -514.912,Z 443.100,A 0.000,B 0.000,C 90.000,E1 53.989} C_DIS
LIN {X -0.281,Y -515.124,Z 443.093,A 0.000,B 0.000,C 90.000,E1 52.844} C_DIS
LIN {X 0.301,Y -515.181,Z 443.090,A 0.000,B 0.000,C 90.000,E1 52.190} C_DIS
LIN {X 0.088,Y -514.957,Z 443.085,A 0.000,B 0.000,C 90.000,E1 51.331} C_DIS
LIN {X 0.118,Y -514.359,Z 443.079,A 0.000,B 0.000,C 90.000,E1 50.150} C_DIS
LIN {X 0.002,Y -513.217,Z 443.071,A 0.000,B 0.000,C 90.000,E1 48.690} C_DIS
LIN {X 0.124,Y -511.614,Z 443.061,A 0.000,B 0.000,C 90.000,E1 46.905} C_DIS
LIN {X 0.059,Y -510.383,Z 443.054,A 0.000,B 0.000,C 90.000,E1 45.729} C_DIS
LIN {X -0.142,Y -508.039,Z 443.041,A 0.000,B 0.000,C 90.000,E1 43.380} C_DIS
LIN {X -0.251,Y -505.987,Z 443.029,A 0.000,B 0.000,C 90.000,E1 41.310} C_DIS
LIN {X -0.131,Y -504.498,Z 443.021,A 0.000,B 0.000,C 90.000,E1 39.806} C_DIS
LIN {X -0.160,Y -502.735,Z 443.011,A 0.000,B 0.000,C 90.000,E1 38.016} C_DIS
LIN {X -0.031,Y -501.203,Z 443.003,A 0.000,B 0.000,C 90.000,E1 36.503} C_DIS
LIN {X 0.017,Y -500.163,Z 442.998,A 0.000,B 0.000,C 90.000,E1 35.598} C_DIS
LIN {X -0.199,Y -498.422,Z 442.989,A 0.000,B 0.000,C 90.000,E1 34.119} C_DIS
LIN {X -0.044,Y -496.594,Z 442.981,A 0.000,B 0.000,C 90.000,E1 32.594} C_DIS
LIN {X -0.032,Y -494.633,Z 442.973,A 0.000,B 0.000,C 90.000,E1 31.082} C_DIS
LIN {X 0.054,Y -491.848,Z 442.961,A 0.000,B 0.000,C 90.000,E1 28.949} C_DIS
LIN {X 0.261,Y -488.757,Z 442.947,A 0.000,B 0.000,C 90.000,E1 26.488} C_DIS
LIN {X -0.090,Y -486.672,Z 442.937,A 0.000,B 0.000,C 90.000,E1 24.695} C_DIS
LIN {X -0.027,Y -485.474,Z 442.930,A 0.000,B 0.000,C 90.000,E1 23.462} C_DIS
LIN {X 0.082,Y -483.241,Z 442.915,A 0.000,B 0.000,C 90.000,E1 20.684} C_DIS
LIN {X -0.061,Y -481.870,Z 442.903,A 0.000,B 0.000,C 90.000,E1 18.544} C_DIS
LIN {X 0.223,Y -481.015,Z 442.896,A 0.000,B 0.000,C 90.000,E1 17.275} C_DIS
LIN {X -0.260,Y -479.976,Z 442.888,A 0.000,B 0.000,C 90.000,E1 15.788} C_DIS
LIN {X 0.137,Y -478.703,Z 442.877,A 0.000,B 0.000,C 90.000,E1 13.883} C_DIS
LIN {X 0.130,Y -477.123,Z 442.860,A 0.000,B 0.000,C 90.000,E1 10.782} C_DIS
LIN {X -0.251,Y -476.370,Z 442.846,A 0.000,B 0.000,C 90.000,E1 8.341} C_DIS
LIN {X -0.090,Y -476.155,Z 442.834,A 0.000,B 0.000,C 90.000,E1 6.144} C_DIS
LIN {X 0.179,Y -476.269,Z 442.824,A 0.000,B 0.000,C 90.000,E1 4.245} C_DIS
LIN {X 0.093,Y -477.362,Z 442.806,A 0.000,B 0.000,C 90.000,E1 1.146} C_DIS
LIN {X -0.230,Y -479.890,Z 442.787,A 0.000,B 0.000,C 90.000,E1 357.650} C_DIS
LIN {X 0.101,Y -481.869,Z 442.777,A 0.000,B 0.000,C 90.000,E1 355.755} C_DIS
LIN {X -0.008,Y -485.433,Z 442.761,A 0.000,B 0.000,C 90.000,E1 352.996} C_DIS
LIN {X -0.114,Y -489.119,Z 442.747,A 0.000,B 0.000,C 90.000,E1 350.557} C_DIS
LIN {X -0.002,Y -492.711,Z 442.736,A 0.000,B 0.000,C 90.000,E1 348.409} C_DIS
LIN {X -0.199,Y -499.381,Z 442.717,A 0.000,B 0.000,C 90.000,E1 345.102} C_DIS
LIN {X 0.148,Y -504.356,Z 442.705,A 0.000,B 0.000,C 90.000,E1 342.960} C_DIS
LIN {X 0.054,Y -512.767,Z 442.687,A 0.000,B 0.000,C 90.000,E1 339.699} C_DIS
LIN {X 0.129,Y -517.502,Z 442.677,A 0.000,B 0.000,C 90.000,E1 337.922} C_DIS
LIN {X -0.127,Y -521.499,Z 442.669,A 0.000,B 0.000,C 90.000,E1 336.485} C_DIS
LIN {X 0.006,Y -524.702,Z 442.663,A 0.000,B 0.000,C 90.000,E1 335.305} C_DIS
LIN {X 0.027,Y -529.527,Z 442.653,A 0.000,B 0.000,C 90.000,E1 333.563} C_DIS
LIN {X -0.080,Y -534.349,Z 442.644,A 0.000,B 0.000,C 90.000,E1 331.847} C_DIS
LIN {X -0.233,Y -537.607,Z 442.637,A 0.000,B 0.000,C 90.000,E1 330.717} C_DIS
LIN {X -0.130,Y -542.555,Z 442.628,A 0.000,B 0.000,C 90.000,E1 328.997} C_DIS
LIN {X -0.099,Y -547.468,Z 442.618,A 0.000,B 0.000,C 90.000,E1 327.296} C_DIS
LIN {X 0.095,Y -553.018,Z 442.607,A 0.000,B 0.000,C 90.000,E1 325.308} C_DIS
LIN {X 0.205,Y -557.866,Z 442.598,A 0.000,B 0.000,C 90.000,E1 323.623} C_DIS
LIN {X 0.058,Y -563.643,Z 442.587,A 0.000,B 0.000,C 90.000,E1 321.698} C_DIS
LIN {X 0.004,Y -570.584,Z 442.575,A 0.000,B 0.000,C 90.000,E1 319.504} C_DIS
LIN {X -0.213,Y -574.976,Z 442.568,A 0.000,B 0.000,C 90.000,E1 318.162} C_DIS
LIN {X -0.263,Y -580.019,Z 442.558,A 0.000,B 0.000,C 90.000,E1 316.539} C_DIS
LIN {X 0.087,Y -586.778,Z 442.547,A 0.000,B 0.000,C 90.000,E1 314.352} C_DIS
LIN {X 0.056,Y -592.810,Z 442.536,A 0.000,B 0.000,C 90.000,E1 312.486} C_DIS
LIN {X -0.044,Y -596.194,Z 442.530,A 0.000,B 0.000,C 90.000,E1 311.434} C_DIS
LIN {X 0.181,Y -600.350,Z 442.523,A 0.000,B 0.000,C 90.000,E1 310.092} C_DIS
LIN {X -0.110,Y -605.191,Z 442.514,A 0.000,B 0.000,C 90.000,E1 308.543} C_DIS
LIN {X 0.174,Y -609.835,Z 442.505,A 0.000,B 0.000,C 90.000,E1 306.950} C_DIS
LIN {X 0.188,Y -614.345,Z 442.497,A 0.000,B 0.000,C 90.000,E1 305.391} C_DIS
LIN {X 0.228,Y -616.494,Z 442.492,A 0.000,B 0.000,C 90.000,E1 304.612} C_DIS
LIN {X -0.297,Y -619.973,Z 442.485,A 0.000,B 0.000,C 90.000,E1 303.372} C_DIS
LIN {X -0.244,Y -623.286,Z 442.478,A 0.000,B 0.000,C 90.000,E1 302.084} C_DIS
LIN {X -0.137,Y -626.456,Z 442.471,A 0.000,B 0.000,C 90.000,E1 300.797} C_DIS
LIN {X 0.226,Y -628.906,Z 442.465,A 0.000,B 0.000,C 90.000,E1 299.745} C_DIS
LIN {X 0.102,Y -631.793,Z 442.458,A 0.000,B 0.000,C 90.000,E1 298.487} C_DIS
LIN {X -0.241,Y -635.197,Z 442.450,A 0.000,B 0.000,C 90.000,E1 297.001} C_DIS
LIN {X -0.004,Y -637.899,Z 442.443,A 0.000,B 0.000,C 90.000,E1 295.720} C_DIS
LIN {X -0.054,Y -639.918,Z 442.437,A 0.000,B 0.000,C 90.000,E1 294.719} C_DIS
LIN {X 0.057,Y -642.689,Z 442.429,A 0.000,B 0.000,C 90.000,E1 293.206} C_DIS
LIN {X -0.037,Y -645.145,Z 442.421,A 0.000,B 0.000,C 90.000,E1 291.716} C_DIS
LIN {X -0.164,Y -647.013,Z 442.414,A 0.000,B 0.000,C 90.000,E1 290.482} C_DIS
LIN {X 0.271,Y -648.418,Z 442.408,A 0.000,B 0.000,C 90.000,E1 289.450} C_DIS
LIN {X -0.031,Y -650.016,Z 442.401,A 0.000,B 0.000,C 90.000,E1 288.236} C_DIS
LIN {X 0.114,Y -651.333,Z 442.394,A 0.000,B 0.000,C 90.000,E1 286.985} C_DIS
LIN {X 0.342,Y -652.706,Z 442.386,A 0.000,B 0.000,C 90.000,E1 285.481} C_DIS
LIN {X -0.027,Y -653.267,Z 442.382,A 0.000,B 0.000,C 90.000,E1 284.773} C_DIS
LIN {X -0.111,Y -654.046,Z 442.374,A 0.000,B 0.000,C 90.000,E1 283.300} C_DIS
LIN {X -0.064,Y -654.478,Z 442.367,A 0.000,B 0.000,C 90.000,E1 282.063} C_DIS
LIN {X -0.269,Y -654.772,Z 442.359,A 0.000,B 0.000,C 90.000,E1 280.602} C_DIS
LIN {X -0.105,Y -654.667,Z 442.355,A 0.000,B 0.000,C 90.000,E1 279.849} C_DIS
LIN {X -0.193,Y -654.326,Z 442.348,A 0.000,B 0.000,C 90.000,E1 278.624} C_DIS
LIN {X 0.255,Y -653.665,Z 442.341,A 0.000,B 0.000,C 90.000,E1 277.352} C_DIS
LIN {X -0.322,Y -653.124,Z 442.337,A 0.000,B 0.000,C 90.000,E1 276.663} C_DIS
LIN {X 0.252,Y -652.182,Z 442.331,A 0.000,B 0.000,C 90.000,E1 275.625} C_DIS
LIN {X -0.058,Y -650.603,Z 442.325,A 0.000,B 0.000,C 90.000,E1 274.416} C_DIS
LIN {X 0.208,Y -648.638,Z 442.318,A 0.000,B 0.000,C 90.000,E1 273.154} C_DIS
LIN {X -0.200,Y -646.444,Z 442.311,A 0.000,B 0.000,C 90.000,E1 271.949} C_DIS
LIN {X 0.218,Y -644.466,Z 442.305,A 0.000,B 0.000,C 90.000,E1 270.917} C_DIS
LIN {X -0.280,Y -641.718,Z 442.298,A 0.000,B 0.000,C 90.000,E1 269.714} C_DIS
LIN {X 0.296,Y -639.985,Z 442.294,A 0.000,B 0.000,C 90.000,E1 268.912} C_DIS
LIN {X -0.015,Y -637.468,Z 442.289,A 0.000,B 0.000,C 90.000,E1 267.936} C_DIS
LIN {X 0.253,Y -634.814,Z 442.283,A 0.000,B 0.000,C 90.000,E1 266.906} C_DIS
LIN {X 0.012,Y -630.746,Z 442.275,A 0.000,B 0.000,C 90.000,E1 265.412} C_DIS
LIN {X -0.242,Y -626.565,Z 442.266,A 0.000,B 0.000,C 90.000,E1 263.913} C_DIS
LIN {X -0.039,Y -623.756,Z 442.260,A 0.000,B 0.000,C 90.000,E1 262.875} C_DIS
LIN {X -0.110,Y -620.080,Z 442.253,A 0.000,B 0.000,C 90.000,E1 261.602} C_DIS
LIN {X 0.090,Y -617.088,Z 442.248,A 0.000,B 0.000,C 90.000,E1 260.557} C_DIS
LIN {X 0.247,Y -614.016,Z 442.242,A 0.000,B 0.000,C 90.000,E1 259.511} C_DIS
LIN {X 0.104,Y -610.102,Z 442.235,A 0.000,B 0.000,C 90.000,E1 258.229} C_DIS
LIN {X 0.019,Y -606.019,Z 442.227,A 0.000,B 0.000,C 90.000,E1 256.937} C_DIS
LIN {X -0.138,Y -601.878,Z 442.220,A 0.000,B 0.000,C 90.000,E1 255.644} C_DIS
LIN {X 0.067,Y -596.648,Z 442.211,A 0.000,B 0.000,C 90.000,E1 254.047} C_DIS
LIN {X 0.060,Y -592.245,Z 442.204,A 0.000,B 0.000,C 90.000,E1 252.725} C_DIS
LIN {X -0.018,Y -587.735,Z 442.197,A 0.000,B 0.000,C 90.000,E1 251.402} C_DIS
LIN {X -0.061,Y -584.982,Z 442.192,A 0.000,B 0.000,C 90.000,E1 250.604} C_DIS
LIN {X -0.070,Y -580.270,Z 442.185,A 0.000,B 0.000,C 90.000,E1 249.263} C_DIS
LIN {X -0.182,Y -577.342,Z 442.180,A 0.000,B 0.000,C 90.000,E1 248.465} C_DIS
LIN {X -0.116,Y -572.321,Z 442.173,A 0.000,B 0.000,C 90.000,E1 247.102} C_DIS
LIN {X 0.030,Y -568.141,Z 442.167,A 0.000,B 0.000,C 90.000,E1 245.997} C_DIS
LIN {X 0.197,Y -561.774,Z 442.158,A 0.000,B 0.000,C 90.000,E1 244.332} C_DIS
LIN {X -0.297,Y -556.365,Z 442.150,A 0.000,B 0.000,C 90.000,E1 242.999} C_DIS
LIN {X 0.116,Y -550.973,Z 442.142,A 0.000,B 0.000,C 90.000,E1 241.563} C_DIS
LIN {X 0.179,Y -544.680,Z 442.133,A 0.000,B 0.000,C 90.000,E1 239.871} C_DIS
LIN {X -0.096,Y -538.484,Z 442.123,A 0.000,B 0.000,C 90.000,E1 238.201} C_DIS
LIN {X 0.083,Y -533.298,Z 442.115,A 0.000,B 0.000,C 90.000,E1 236.755} C_DIS
LIN {X 0.170,Y -528.058,Z 442.107,A 0.000,B 0.000,C 90.000,E1 235.308} C_DIS
LIN {X 0.111,Y -521.900,Z 442.098,A 0.000,B 0.000,C 90.000,E1 233.577} C_DIS
LIN {X 0.115,Y -515.922,Z 442.088,A 0.000,B 0.000,C 90.000,E1 231.823} C_DIS
LIN {X 0.276,Y -506.667,Z 442.072,A 0.000,B 0.000,C 90.000,E1 228.852} C_DIS
LIN {X 0.098,Y -500.545,Z 442.060,A 0.000,B 0.000,C 90.000,E1 226.782} C_DIS
LIN {X 0.086,Y -494.580,Z 442.048,A 0.000,B 0.000,C 90.000,E1 224.676} C_DIS
LIN {X 0.275,Y -488.742,Z 442.036,A 0.000,B 0.000,C 90.000,E1 222.528} C_DIS
LIN {X 0.018,Y -483.174,Z 442.025,A 0.000,B 0.000,C 90.000,E1 220.415} C_DIS
LIN {X -0.006,Y -477.805,Z 442.013,A 0.000,B 0.000,C 90.000,E1 218.257} C_DIS
LIN {X 0.071,Y -469.858,Z 441.994,A 0.000,B 0.000,C 90.000,E1 214.818} C_DIS
LIN {X 0.083,Y -466.428,Z 441.985,A 0.000,B 0.000,C 90.000,E1 213.245} C_DIS
LIN {X -0.089,Y -461.733,Z 441.973,A 0.000,B 0.000,C 90.000,E1 211.052} C_DIS
LIN {X -0.085,Y -458.467,Z 441.964,A 0.000,B 0.000,C 90.000,E1 209.461} C_DIS
LIN {X 0.139,Y -454.540,Z 441.953,A 0.000,B 0.000,C 90.000,E1 207.513} C_DIS
LIN {X 0.062,Y -450.503,Z 441.942,A 0.000,B 0.000,C 90.000,E1 205.591} C_DIS
LIN {X 0.106,Y -446.428,Z 441.931,A 0.000,B 0.000,C 90.000,E1 203.643} C_DIS
LIN {X 0.003,Y -441.009,Z 441.917,A 0.000,B 0.000,C 90.000,E1 201.046} C_DIS
LIN {X 0.065,Y -437.809,Z 441.908,A 0.000,B 0.000,C 90.000,E1 199.396} C_DIS
LIN {X 0.208,Y -433.083,Z 441.893,A 0.000,B 0.000,C 90.000,E1 196.732} C_DIS
LIN {X 0.035,Y -429.269,Z 441.880,A 0.000,B 0.000,C 90.000,E1 194.426} C_DIS
LIN {X -0.055,Y -424.728,Z 441.863,A 0.000,B 0.000,C 90.000,E1 191.422} C_DIS
LIN {X -0.140,Y -420.734,Z 441.847,A 0.000,B 0.000,C 90.000,E1 188.398} C_DIS
LIN {X 0.152,Y -418.754,Z 441.837,A 0.000,B 0.000,C 90.000,E1 186.663} C_DIS
LIN {X -0.063,Y -416.904,Z 441.828,A 0.000,B 0.000,C 90.000,E1 184.992} C_DIS
LIN {X 0.124,Y -414.322,Z 441.813,A 0.000,B 0.000,C 90.000,E1 182.236} C_DIS
LIN {X 0.196,Y -412.065,Z 441.795,A 0.000,B 0.000,C 90.000,E1 179.141} C_DIS
LIN {X -0.205,Y -410.660,Z 441.778,A 0.000,B 0.000,C 90.000,E1 176.102} C_DIS
LIN {X -0.028,Y -410.313,Z 441.751,A 0.000,B 0.000,C 90.000,E1 171.254} C_DIS
LIN {X -0.023,Y -411.341,Z 441.730,A 0.000,B 0.000,C 90.000,E1 167.465} C_DIS
LIN {X 0.090,Y -412.863,Z 441.715,A 0.000,B 0.000,C 90.000,E1 164.700} C_DIS
LIN {X -0.014,Y -416.260,Z 441.692,A 0.000,B 0.000,C 90.000,E1 160.604} C_DIS
LIN {X -0.083,Y -420.528,Z 441.671,A 0.000,B 0.000,C 90.000,E1 156.869} C_DIS
LIN {X -0.007,Y -424.168,Z 441.656,A 0.000,B 0.000,C 90.000,E1 154.152} C_DIS
LIN {X -0.020,Y -428.850,Z 441.640,A 0.000,B 0.000,C 90.000,E1 151.129} C_DIS
LIN {X -0.019,Y -432.142,Z 441.629,A 0.000,B 0.000,C 90.000,E1 149.125} C_DIS
LIN {X -0.258,Y -436.947,Z 441.614,A 0.000,B 0.000,C 90.000,E1 146.501} C_DIS
LIN {X 0.049,Y -440.791,Z 441.603,A 0.000,B 0.000,C 90.000,E1 144.482} C_DIS
LIN {X -0.267,Y -446.271,Z 441.588,A 0.000,B 0.000,C 90.000,E1 141.904} C_DIS
LIN {X 0.093,Y -450.650,Z 441.577,A 0.000,B 0.000,C 90.000,E1 139.908} C_DIS
LIN {X -0.129,Y -455.061,Z 441.567,A 0.000,B 0.000,C 90.000,E1 138.000} C_DIS
LIN {X 0.054,Y -459.308,Z 441.556,A 0.000,B 0.000,C 90.000,E1 136.053} C_DIS
LIN {X 0.271,Y -462.406,Z 441.547,A 0.000,B 0.000,C 90.000,E1 134.433} C_DIS
LIN {X -0.171,Y -464.526,Z 441.540,A 0.000,B 0.000,C 90.000,E1 133.218} C_DIS
LIN {X 0.094,Y -466.210,Z 441.533,A 0.000,B 0.000,C 90.000,E1 131.919} C_DIS
LIN {X 0.036,Y -467.289,Z 441.526,A 0.000,B 0.000,C 90.000,E1 130.663} C_DIS
LIN {X -0.022,Y -467.708,Z 441.521,A 0.000,B 0.000,C 90.000,E1 129.725} C_DIS
LIN {X 0.225,Y -467.568,Z 441.515,A 0.000,B 0.000,C 90.000,E1 128.749} C_DIS
LIN {X 0.177,Y -466.932,Z 441.510,A 0.000,B 0.000,C 90.000,E1 127.810} C_DIS
LIN {X 0.124,Y -465.932,Z 441.505,A 0.000,B 0.000,C 90.000,E1 126.870} C_DIS
LIN {X 0.056,Y -464.530,Z 441.500,A 0.000,B 0.000,C 90.000,E1 125.931} C_DIS
LIN {X -0.054,Y -463.390,Z 441.496,A 0.000,B 0.000,C 90.000,E1 125.311} C_DIS
LIN {X 0.222,Y -461.388,Z 441.491,A 0.000,B 0.000,C 90.000,E1 124.326} C_DIS
LIN {X 0.214,Y -459.017,Z 441.486,A 0.000,B 0.000,C 90.000,E1 123.372} C_DIS
LIN {X -0.092,Y -455.387,Z 441.479,A 0.000,B 0.000,C 90.000,E1 122.133} C_DIS
LIN {X 0.016,Y -450.329,Z 441.470,A 0.000,B 0.000,C 90.000,E1 120.512} C_DIS
LIN {X 0.038,Y -447.095,Z 441.464,A 0.000,B 0.000,C 90.000,E1 119.539} C_DIS
LIN {X 0.141,Y -441.404,Z 441.455,A 0.000,B 0.000,C 90.000,E1 117.897} C_DIS
LIN {X -0.172,Y -438.521,Z 441.451,A 0.000,B 0.000,C 90.000,E1 117.129} C_DIS
LIN {X -0.211,Y -438.534,Z 441.451,A 0.000,B 0.000,C 90.000,E1 117.129} C_DIS
LIN {X 0.080,Y -444.691,Z 441.439,A 0.000,B 0.000,C 90.000,E1 114.951} C_DIS
LIN {X 0.052,Y -454.664,Z 441.415,A 0.000,B 0.000,C 90.000,E1 110.737} C_DIS
LIN {X 0.174,Y -457.319,Z 441.410,A 0.000,B 0.000,C 90.000,E1 109.758} C_DIS
LIN {X -0.188,Y -465.943,Z 441.387,A 0.000,B 0.000,C 90.000,E1 105.662} C_DIS
LIN {X -0.016,Y -467.506,Z 441.383,A 0.000,B 0.000,C 90.000,E1 105.009} C_DIS
LIN {X -0.212,Y -468.094,Z 441.382,A 0.000,B 0.000,C 90.000,E1 104.717} C_DIS
LIN {X -0.073,Y -475.750,Z 441.357,A 0.000,B 0.000,C 90.000,E1 100.310} C_DIS
LIN {X 0.233,Y -476.283,Z 441.356,A 0.000,B 0.000,C 90.000,E1 99.962} C_DIS
LIN {X 0.181,Y -481.751,Z 441.331,A 0.000,B 0.000,C 90.000,E1 95.625} C_DIS
LIN {X 0.028,Y -482.162,Z 441.330,A 0.000,B 0.000,C 90.000,E1 95.334} C_DIS
LIN {X -0.218,Y -485.538,Z 441.304,A 0.000,B 0.000,C 90.000,E1 90.745} C_DIS
LIN {X -0.010,Y -486.308,Z 441.282,A 0.000,B 0.000,C 90.000,E1 86.731} C_DIS
LIN {X 0.124,Y -486.322,Z 441.278,A 0.000,B 0.000,C 90.000,E1 86.102} C_DIS
LIN {X 0.197,Y -484.626,Z 441.253,A 0.000,B 0.000,C 90.000,E1 81.489} C_DIS
LIN {X 0.077,Y -480.554,Z 441.227,A 0.000,B 0.000,C 90.000,E1 76.881} C_DIS
LIN {X -0.013,Y -474.309,Z 441.201,A 0.000,B 0.000,C 90.000,E1 72.236} C_DIS
LIN {X -0.192,Y -473.898,Z 441.200,A 0.000,B 0.000,C 90.000,E1 71.945} C_DIS
LIN {X -0.066,Y -466.289,Z 441.175,A 0.000,B 0.000,C 90.000,E1 67.539} C_DIS
LIN {X -0.122,Y -465.859,Z 441.173,A 0.000,B 0.000,C 90.000,E1 67.230} C_DIS
LIN {X -0.180,Y -465.291,Z 441.172,A 0.000,B 0.000,C 90.000,E1 66.922} C_DIS
LIN {X 0.016,Y -462.664,Z 441.165,A 0.000,B 0.000,C 90.000,E1 65.741} C_DIS
LIN {X -0.024,Y -462.697,Z 441.165,A 0.000,B 0.000,C 90.000,E1 65.741} C_DIS
LIN {X 0.080,Y -473.769,Z 441.157,A 0.000,B 0.000,C 90.000,E1 64.204} C_DIS
LIN {X -0.257,Y -482.755,Z 441.150,A 0.000,B 0.000,C 90.000,E1 62.999} C_DIS
LIN {X -0.271,Y -488.054,Z 441.146,A 0.000,B 0.000,C 90.000,E1 62.231} C_DIS
LIN {X -0.028,Y -491.968,Z 441.142,A 0.000,B 0.000,C 90.000,E1 61.591} C_DIS
LIN {X 0.052,Y -495.702,Z 441.139,A 0.000,B 0.000,C 90.000,E1 60.973} C_DIS
LIN {X -0.120,Y -498.351,Z 441.136,A 0.000,B 0.000,C 90.000,E1 60.539} C_DIS
LIN {X 0.016,Y -501.525,Z 441.133,A 0.000,B 0.000,C 90.000,E1 59.921} C_DIS
LIN {X -0.265,Y -504.989,Z 441.129,A 0.000,B 0.000,C 90.000,E1 59.203} C_DIS
LIN {X -0.068,Y -507.459,Z 441.125,A 0.000,B 0.000,C 90.000,E1 58.584} C_DIS
LIN {X -0.120,Y -509.602,Z 441.122,A 0.000,B 0.000,C 90.000,E1 57.995} C_DIS
LIN {X 0.113,Y -511.338,Z 441.119,A 0.000,B 0.000,C 90.000,E1 57.375} C_DIS
LIN {X 0.082,Y -512.789,Z 441.116,A 0.000,B 0.000,C 90.000,E1 56.786} C_DIS
LIN {X -0.004,Y -513.482,Z 441.114,A 0.000,B 0.000,C 90.000,E1 56.501} C_DIS
LIN {X 0.185,Y -515.024,Z 441.109,A 0.000,B 0.000,C 90.000,E1 55.595} C_DIS
LIN {X -0.029,Y -515.978,Z 441.104,A 0.000,B 0.000,C 90.000,E1 54.736} C_DIS
LIN {X 0.257,Y -516.377,Z 441.101,A 0.000,B 0.000,C 90.000,E1 54.116} C_DIS
LIN {X 0.062,Y -516.596,Z 441.096,A 0.000,B 0.000,C 90.000,E1 53.256} C_DIS
LIN {X -0.129,Y -516.660,Z 441.091,A 0.000,B 0.000,C 90.000,E1 52.396} C_DIS
LIN {X -0.323,Y -516.455,Z 441.086,A 0.000,B 0.000,C 90.000,E1 51.537} C_DIS
LIN {X -0.267,Y -515.801,Z 441.080,A 0.000,B 0.000,C 90.000,E1 50.356} C_DIS
LIN {X 0.112,Y -514.899,Z 441.073,A 0.000,B 0.000,C 90.000,E1 49.138} C_DIS
LIN {X 0.014,Y -513.519,Z 441.065,A 0.000,B 0.000,C 90.000,E1 47.676} C_DIS
LIN {X -0.019,Y -512.352,Z 441.058,A 0.000,B 0.000,C 90.000,E1 46.500} C_DIS
LIN {X -0.040,Y -510.127,Z 441.047,A 0.000,B 0.000,C 90.000,E1 44.433} C_DIS
LIN {X -0.126,Y -508.974,Z 441.040,A 0.000,B 0.000,C 90.000,E1 43.257} C_DIS
LIN {X 0.134,Y -506.903,Z 441.029,A 0.000,B 0.000,C 90.000,E1 41.148} C_DIS
LIN {X 0.055,Y -504.780,Z 441.017,A 0.000,B 0.000,C 90.000,E1 39.072} C_DIS
LIN {X -0.168,Y -503.285,Z 441.009,A 0.000,B 0.000,C 90.000,E1 37.604} C_DIS
LIN {X -0.024,Y -501.714,Z 441.001,A 0.000,B 0.000,C 90.000,E1 36.091} C_DIS
LIN {X 0.078,Y -499.602,Z 440.991,A 0.000,B 0.000,C 90.000,E1 34.278} C_DIS
LIN {X 0.125,Y -497.344,Z 440.980,A 0.000,B 0.000,C 90.000,E1 32.467} C_DIS
LIN {X -0.271,Y -495.391,Z 440.972,A 0.000,B 0.000,C 90.000,E1 31.003} C_DIS
LIN {X -0.001,Y -493.001,Z 440.962,A 0.000,B 0.000,C 90.000,E1 29.155} C_DIS
LIN {X -0.189,Y -489.885,Z 440.949,A 0.000,B 0.000,C 90.000,E1 26.744} C_DIS
LIN {X 0.191,Y -486.874,Z 440.933,A 0.000,B 0.000,C 90.000,E1 23.951} C_DIS
LIN {X -0.095,Y -484.042,Z 440.914,A 0.000,B 0.000,C 90.000,E1 20.610} C_DIS
LIN {X 0.231,Y -482.659,Z 440.903,A 0.000,B 0.000,C 90.000,E1 18.417} C_DIS
LIN {X -0.079,Y -481.834,Z 440.896,A 0.000,B 0.000,C 90.000,E1 17.221} C_DIS
LIN {X -0.097,Y -480.559,Z 440.885,A 0.000,B 0.000,C 90.000,E1 15.371} C_DIS
LIN {X 0.010,Y -478.948,Z 440.872,A 0.000,B 0.000,C 90.000,E1 12.883} C_DIS
LIN {X -0.157,Y -477.830,Z 440.858,A 0.000,B 0.000,C 90.000,E1 10.423} C_DIS
LIN {X 0.186,Y -477.116,Z 440.842,A 0.000,B 0.000,C 90.000,E1 7.587} C_DIS
LIN {X 0.238,Y -477.088,Z 440.825,A 0.000,B 0.000,C 90.000,E1 4.473} C_DIS
LIN {X -0.223,Y -478.394,Z 440.804,A 0.000,B 0.000,C 90.000,E1 0.802} C_DIS
LIN {X 0.141,Y -482.713,Z 440.777,A 0.000,B 0.000,C 90.000,E1 355.755} C_DIS
LIN {X 0.063,Y -486.328,Z 440.761,A 0.000,B 0.000,C 90.000,E1 352.996} C_DIS
LIN {X -0.016,Y -490.052,Z 440.748,A 0.000,B 0.000,C 90.000,E1 350.557} C_DIS
LIN {X 0.023,Y -494.198,Z 440.734,A 0.000,B 0.000,C 90.000,E1 348.117} C_DIS
LIN {X -0.034,Y -500.338,Z 440.717,A 0.000,B 0.000,C 90.000,E1 345.102} C_DIS
LIN {X -0.144,Y -505.305,Z 440.706,A 0.000,B 0.000,C 90.000,E1 343.015} C_DIS
LIN {X 0.173,Y -512.903,Z 440.689,A 0.000,B 0.000,C 90.000,E1 340.007} C_DIS
LIN {X 0.120,Y -516.872,Z 440.681,A 0.000,B 0.000,C 90.000,E1 338.539} C_DIS
LIN {X 0.000,Y -521.690,Z 440.671,A 0.000,B 0.000,C 90.000,E1 336.794} C_DIS
LIN {X -0.178,Y -525.708,Z 440.663,A 0.000,B 0.000,C 90.000,E1 335.357} C_DIS
LIN {X 0.109,Y -530.533,Z 440.653,A 0.000,B 0.000,C 90.000,E1 333.589} C_DIS
LIN {X -0.022,Y -536.219,Z 440.642,A 0.000,B 0.000,C 90.000,E1 331.591} C_DIS
LIN {X -0.148,Y -539.520,Z 440.636,A 0.000,B 0.000,C 90.000,E1 330.461} C_DIS
LIN {X 0.258,Y -543.698,Z 440.628,A 0.000,B 0.000,C 90.000,E1 328.997} C_DIS
LIN {X 0.020,Y -548.625,Z 440.619,A 0.000,B 0.000,C 90.000,E1 327.327} C_DIS
LIN {X -0.225,Y -554.214,Z 440.608,A 0.000,B 0.000,C 90.000,E1 325.388} C_DIS
LIN {X -0.096,Y -559.103,Z 440.598,A 0.000,B 0.000,C 90.000,E1 323.703} C_DIS
LIN {X 0.026,Y -564.050,Z 440.589,A 0.000,B 0.000,C 90.000,E1 322.029} C_DIS
LIN {X 0.066,Y -571.012,Z 440.577,A 0.000,B 0.000,C 90.000,E1 319.828} C_DIS
LIN {X 0.373,Y -576.303,Z 440.568,A 0.000,B 0.000,C 90.000,E1 318.162} C_DIS
LIN {X 0.085,Y -582.224,Z 440.557,A 0.000,B 0.000,C 90.000,E1 316.296} C_DIS
LIN {X -0.330,Y -589.079,Z 440.545,A 0.000,B 0.000,C 90.000,E1 314.190} C_DIS
LIN {X 0.091,Y -595.159,Z 440.535,A 0.000,B 0.000,C 90.000,E1 312.285} C_DIS
LIN {X -0.155,Y -599.403,Z 440.528,A 0.000,B 0.000,C 90.000,E1 310.987} C_DIS
LIN {X -0.121,Y -602.717,Z 440.522,A 0.000,B 0.000,C 90.000,E1 309.930} C_DIS
LIN {X 0.106,Y -607.626,Z 440.513,A 0.000,B 0.000,C 90.000,E1 308.338} C_DIS
LIN {X -0.044,Y -612.221,Z 440.504,A 0.000,B 0.000,C 90.000,E1 306.790} C_DIS
LIN {X -0.291,Y -616.016,Z 440.497,A 0.000,B 0.000,C 90.000,E1 305.518} C_DIS
LIN {X 0.033,Y -619.599,Z 440.490,A 0.000,B 0.000,C 90.000,E1 304.199} C_DIS
LIN {X 0.081,Y -623.044,Z 440.483,A 0.000,B 0.000,C 90.000,E1 302.911} C_DIS
LIN {X 0.192,Y -625.689,Z 440.477,A 0.000,B 0.000,C 90.000,E1 301.878} C_DIS
LIN {X -0.188,Y -629.487,Z 440.469,A 0.000,B 0.000,C 90.000,E1 300.384} C_DIS
LIN {X 0.213,Y -631.917,Z 440.463,A 0.000,B 0.000,C 90.000,E1 299.333} C_DIS
LIN {X -0.128,Y -635.369,Z 440.455,A 0.000,B 0.000,C 90.000,E1 297.847} C_DIS
LIN {X 0.117,Y -638.208,Z 440.448,A 0.000,B 0.000,C 90.000,E1 296.565} C_DIS
LIN {X -0.167,Y -640.843,Z 440.441,A 0.000,B 0.000,C 90.000,E1 295.335} C_DIS
LIN {X -0.179,Y -642.786,Z 440.435,A 0.000,B 0.000,C 90.000,E1 294.335} C_DIS
LIN {X -0.161,Y -644.705,Z 440.430,A 0.000,B 0.000,C 90.000,E1 293.334} C_DIS
LIN {X -0.213,Y -647.169,Z 440.421,A 0.000,B 0.000,C 90.000,E1 291.844} C_DIS
LIN {X -0.304,Y -649.078,Z 440.414,A 0.000,B 0.000,C 90.000,E1 290.610} C_DIS
LIN {X 0.237,Y -650.848,Z 440.408,A 0.000,B 0.000,C 90.000,E1 289.322} C_DIS
LIN {X -0.102,Y -652.142,Z 440.402,A 0.000,B 0.000,C 90.000,E1 288.362} C_DIS
LIN {X 0.275,Y -653.498,Z 440.395,A 0.000,B 0.000,C 90.000,E1 287.094} C_DIS
LIN {X -0.270,Y -654.869,Z 440.387,A 0.000,B 0.000,C 90.000,E1 285.662} C_DIS
LIN {X -0.049,Y -655.617,Z 440.380,A 0.000,B 0.000,C 90.000,E1 284.411} C_DIS
LIN {X 0.019,Y -656.215,Z 440.373,A 0.000,B 0.000,C 90.000,E1 283.175} C_DIS
LIN {X 0.069,Y -656.583,Z 440.368,A 0.000,B 0.000,C 90.000,E1 282.187} C_DIS
LIN {X 0.037,Y -656.757,Z 440.360,A 0.000,B 0.000,C 90.000,E1 280.715} C_DIS
LIN {X 0.100,Y -656.666,Z 440.354,A 0.000,B 0.000,C 90.000,E1 279.726} C_DIS
LIN {X 0.059,Y -656.414,Z 440.349,A 0.000,B 0.000,C 90.000,E1 278.746} C_DIS
LIN {X -0.097,Y -655.733,Z 440.342,A 0.000,B 0.000,C 90.000,E1 277.530} C_DIS
LIN {X 0.076,Y -655.221,Z 440.338,A 0.000,B 0.000,C 90.000,E1 276.777} C_DIS
LIN {X 0.026,Y -654.264,Z 440.332,A 0.000,B 0.000,C 90.000,E1 275.796} C_DIS
LIN {X -0.253,Y -652.714,Z 440.325,A 0.000,B 0.000,C 90.000,E1 274.588} C_DIS
LIN {X 0.254,Y -651.196,Z 440.320,A 0.000,B 0.000,C 90.000,E1 273.555} C_DIS
LIN {X -0.118,Y -649.069,Z 440.313,A 0.000,B 0.000,C 90.000,E1 272.350} C_DIS
LIN {X 0.118,Y -646.639,Z 440.306,A 0.000,B 0.000,C 90.000,E1 271.088} C_DIS
LIN {X -0.122,Y -644.494,Z 440.301,A 0.000,B 0.000,C 90.000,E1 270.115} C_DIS
LIN {X 0.254,Y -642.233,Z 440.295,A 0.000,B 0.000,C 90.000,E1 269.083} C_DIS
LIN {X -0.266,Y -639.105,Z 440.288,A 0.000,B 0.000,C 90.000,E1 267.879} C_DIS
LIN {X 0.058,Y -636.438,Z 440.283,A 0.000,B 0.000,C 90.000,E1 266.846} C_DIS
LIN {X -0.184,Y -632.317,Z 440.274,A 0.000,B 0.000,C 90.000,E1 265.355} C_DIS
LIN {X -0.191,Y -628.833,Z 440.267,A 0.000,B 0.000,C 90.000,E1 264.090} C_DIS
LIN {X -0.184,Y -625.257,Z 440.260,A 0.000,B 0.000,C 90.000,E1 262.818} C_DIS
LIN {X -0.232,Y -621.561,Z 440.253,A 0.000,B 0.000,C 90.000,E1 261.546} C_DIS
LIN {X -0.013,Y -618.561,Z 440.247,A 0.000,B 0.000,C 90.000,E1 260.500} C_DIS
LIN {X 0.292,Y -613.936,Z 440.239,A 0.000,B 0.000,C 90.000,E1 258.926} C_DIS
LIN {X -0.205,Y -610.696,Z 440.233,A 0.000,B 0.000,C 90.000,E1 257.937} C_DIS
LIN {X -0.279,Y -606.592,Z 440.226,A 0.000,B 0.000,C 90.000,E1 256.645} C_DIS
LIN {X -0.008,Y -603.241,Z 440.220,A 0.000,B 0.000,C 90.000,E1 255.574} C_DIS
LIN {X 0.236,Y -598.000,Z 440.211,A 0.000,B 0.000,C 90.000,E1 253.976} C_DIS
LIN {X 0.083,Y -593.547,Z 440.204,A 0.000,B 0.000,C 90.000,E1 252.670} C_DIS
LIN {X 0.211,Y -589.010,Z 440.196,A 0.000,B 0.000,C 90.000,E1 251.329} C_DIS
LIN {X -0.143,Y -585.300,Z 440.191,A 0.000,B 0.000,C 90.000,E1 250.296} C_DIS
LIN {X -0.001,Y -581.492,Z 440.185,A 0.000,B 0.000,C 90.000,E1 249.209} C_DIS
LIN {X -0.103,Y -578.539,Z 440.180,A 0.000,B 0.000,C 90.000,E1 248.411} C_DIS
LIN {X -0.023,Y -573.498,Z 440.173,A 0.000,B 0.000,C 90.000,E1 247.050} C_DIS
LIN {X -0.153,Y -569.291,Z 440.166,A 0.000,B 0.000,C 90.000,E1 245.973} C_DIS
LIN {X -0.003,Y -563.980,Z 440.159,A 0.000,B 0.000,C 90.000,E1 244.588} C_DIS
LIN {X 0.040,Y -558.547,Z 440.151,A 0.000,B 0.000,C 90.000,E1 243.204} C_DIS
LIN {X -0.005,Y -553.148,Z 440.143,A 0.000,B 0.000,C 90.000,E1 241.820} C_DIS
LIN {X -0.134,Y -545.761,Z 440.133,A 0.000,B 0.000,C 90.000,E1 239.871} C_DIS
LIN {X 0.086,Y -538.494,Z 440.122,A 0.000,B 0.000,C 90.000,E1 237.867} C_DIS
LIN {X 0.262,Y -533.327,Z 440.114,A 0.000,B 0.000,C 90.000,E1 236.421} C_DIS
LIN {X 0.297,Y -526.023,Z 440.102,A 0.000,B 0.000,C 90.000,E1 234.402} C_DIS
LIN {X -0.147,Y -521.976,Z 440.096,A 0.000,B 0.000,C 90.000,E1 233.290} C_DIS
LIN {X -0.076,Y -517.018,Z 440.088,A 0.000,B 0.000,C 90.000,E1 231.823} C_DIS
LIN {X 0.028,Y -506.844,Z 440.070,A 0.000,B 0.000,C 90.000,E1 228.566} C_DIS
LIN {X 0.192,Y -500.759,Z 440.058,A 0.000,B 0.000,C 90.000,E1 226.458} C_DIS
LIN {X -0.003,Y -495.667,Z 440.048,A 0.000,B 0.000,C 90.000,E1 224.676} C_DIS
LIN {X 0.215,Y -489.820,Z 440.036,A 0.000,B 0.000,C 90.000,E1 222.528} C_DIS
LIN {X 0.162,Y -485.015,Z 440.026,A 0.000,B 0.000,C 90.000,E1 220.701} C_DIS
LIN {X 0.180,Y -479.587,Z 440.014,A 0.000,B 0.000,C 90.000,E1 218.543} C_DIS
LIN {X 0.160,Y -472.233,Z 439.997,A 0.000,B 0.000,C 90.000,E1 215.438} C_DIS
LIN {X -0.018,Y -468.105,Z 439.987,A 0.000,B 0.000,C 90.000,E1 213.579} C_DIS
LIN {X 0.106,Y -464.022,Z 439.976,A 0.000,B 0.000,C 90.000,E1 211.671} C_DIS
LIN {X 0.160,Y -460.696,Z 439.967,A 0.000,B 0.000,C 90.000,E1 210.079} C_DIS
LIN {X 0.032,Y -458.069,Z 439.960,A 0.000,B 0.000,C 90.000,E1 208.821} C_DIS
LIN {X 0.151,Y -454.737,Z 439.951,A 0.000,B 0.000,C 90.000,E1 207.206} C_DIS
LIN {X 0.201,Y -451.368,Z 439.942,A 0.000,B 0.000,C 90.000,E1 205.591} C_DIS
LIN {X -0.145,Y -447.269,Z 439.932,A 0.000,B 0.000,C 90.000,E1 203.695} C_DIS
LIN {X 0.055,Y -443.133,Z 439.921,A 0.000,B 0.000,C 90.000,E1 201.716} C_DIS
LIN {X 0.155,Y -439.879,Z 439.912,A 0.000,B 0.000,C 90.000,E1 200.066} C_DIS
LIN {X 0.192,Y -434.398,Z 439.895,A 0.000,B 0.000,C 90.000,E1 197.094} C_DIS
LIN {X -0.146,Y -429.967,Z 439.880,A 0.000,B 0.000,C 90.000,E1 194.481} C_DIS
LIN {X -0.215,Y -425.386,Z 439.864,A 0.000,B 0.000,C 90.000,E1 191.478} C_DIS
LIN {X -0.203,Y -420.972,Z 439.845,A 0.000,B 0.000,C 90.000,E1 188.106} C_DIS
LIN {X 0.089,Y -418.987,Z 439.836,A 0.000,B 0.000,C 90.000,E1 186.372} C_DIS
LIN {X -0.179,Y -417.506,Z 439.828,A 0.000,B 0.000,C 90.000,E1 185.049} C_DIS
LIN {X 0.065,Y -414.357,Z 439.809,A 0.000,B 0.000,C 90.000,E1 181.604} C_DIS
LIN {X 0.129,Y -412.250,Z 439.792,A 0.000,B 0.000,C 90.000,E1 178.511} C_DIS
LIN {X 0.164,Y -411.046,Z 439.775,A 0.000,B 0.000,C 90.000,E1 175.412} C_DIS
LIN {X -0.078,Y -410.897,Z 439.750,A 0.000,B 0.000,C 90.000,E1 170.971} C_DIS
LIN {X -0.129,Y -411.738,Z 439.733,A 0.000,B 0.000,C 90.000,E1 167.881} C_DIS
LIN {X 0.097,Y -413.188,Z 439.717,A 0.000,B 0.000,C 90.000,E1 165.102} C_DIS
LIN {X -0.233,Y -416.492,Z 439.695,A 0.000,B 0.000,C 90.000,E1 161.040} C_DIS
LIN {X -0.097,Y -418.195,Z 439.685,A 0.000,B 0.000,C 90.000,E1 159.316} C_DIS
LIN {X -0.200,Y -421.550,Z 439.670,A 0.000,B 0.000,C 90.000,E1 156.613} C_DIS
LIN {X 0.128,Y -424.761,Z 439.657,A 0.000,B 0.000,C 90.000,E1 154.204} C_DIS
LIN {X 0.149,Y -429.479,Z 439.640,A 0.000,B 0.000,C 90.000,E1 151.179} C_DIS
LIN {X -0.022,Y -434.020,Z 439.625,A 0.000,B 0.000,C 90.000,E1 148.535} C_DIS
LIN {X 0.029,Y -439.027,Z 439.611,A 0.000,B 0.000,C 90.000,E1 145.881} C_DIS
LIN {X 0.017,Y -444.363,Z 439.596,A 0.000,B 0.000,C 90.000,E1 143.256} C_DIS
LIN {X 0.111,Y -449.448,Z 439.583,A 0.000,B 0.000,C 90.000,E1 140.964} C_DIS
LIN {X -0.150,Y -453.214,Z 439.574,A 0.000,B 0.000,C 90.000,E1 139.380} C_DIS
LIN {X -0.035,Y -456.977,Z 439.565,A 0.000,B 0.000,C 90.000,E1 137.757} C_DIS
LIN {X 0.154,Y -460.578,Z 439.556,A 0.000,B 0.000,C 90.000,E1 136.134} C_DIS
LIN {X 0.244,Y -461.921,Z 439.553,A 0.000,B 0.000,C 90.000,E1 135.486} C_DIS
LIN {X -0.201,Y -464.427,Z 439.546,A 0.000,B 0.000,C 90.000,E1 134.271} C_DIS
LIN {X -0.021,Y -466.032,Z 439.541,A 0.000,B 0.000,C 90.000,E1 133.299} C_DIS
LIN {X -0.143,Y -467.391,Z 439.535,A 0.000,B 0.000,C 90.000,E1 132.366} C_DIS
LIN {X 0.028,Y -468.210,Z 439.532,A 0.000,B 0.000,C 90.000,E1 131.714} C_DIS
LIN {X 0.004,Y -469.270,Z 439.525,A 0.000,B 0.000,C 90.000,E1 130.458} C_DIS
LIN {X -0.028,Y -469.648,Z 439.520,A 0.000,B 0.000,C 90.000,E1 129.519} C_DIS
LIN {X -0.122,Y -469.432,Z 439.514,A 0.000,B 0.000,C 90.000,E1 128.588} C_DIS
LIN {X -0.151,Y -468.717,Z 439.509,A 0.000,B 0.000,C 90.000,E1 127.649} C_DIS
LIN {X 0.189,Y -467.657,Z 439.504,A 0.000,B 0.000,C 90.000,E1 126.664} C_DIS
LIN {X 0.141,Y -466.196,Z 439.499,A 0.000,B 0.000,C 90.000,E1 125.724} C_DIS
LIN {X -0.196,Y -464.332,Z 439.493,A 0.000,B 0.000,C 90.000,E1 124.818} C_DIS
LIN {X -0.303,Y -462.933,Z 439.490,A 0.000,B 0.000,C 90.000,E1 124.199} C_DIS
LIN {X 0.221,Y -461.342,Z 439.486,A 0.000,B 0.000,C 90.000,E1 123.499} C_DIS
LIN {X 0.062,Y -456.794,Z 439.477,A 0.000,B 0.000,C 90.000,E1 121.926} C_DIS
LIN {X -0.036,Y -451.585,Z 439.469,A 0.000,B 0.000,C 90.000,E1 120.335} C_DIS
LIN {X 0.228,Y -448.255,Z 439.463,A 0.000,B 0.000,C 90.000,E1 119.333} C_DIS
LIN {X 0.082,Y -443.645,Z 439.456,A 0.000,B 0.000,C 90.000,E1 118.052} C_DIS
LIN {X -0.198,Y -439.250,Z 439.449,A 0.000,B 0.000,C 90.000,E1 116.873} C_DIS
LIN {X -0.237,Y -439.239,Z 439.449,A 0.000,B 0.000,C 90.000,E1 116.873} C_DIS
LIN {X 0.072,Y -444.231,Z 439.440,A 0.000,B 0.000,C 90.000,E1 115.103} C_DIS
LIN {X 0.114,Y -445.098,Z 439.438,A 0.000,B 0.000,C 90.000,E1 114.771} C_DIS
LIN {X -0.203,Y -454.263,Z 439.416,A 0.000,B 0.000,C 90.000,E1 110.918} C_DIS
LIN {X -0.087,Y -456.928,Z 439.411,A 0.000,B 0.000,C 90.000,E1 109.939} C_DIS
LIN {X 0.151,Y -458.209,Z 439.407,A 0.000,B 0.000,C 90.000,E1 109.268} C_DIS
LIN {X -0.099,Y -466.357,Z 439.386,A 0.000,B 0.000,C 90.000,E1 105.481} C_DIS
LIN {X 0.074,Y -467.886,Z 439.382,A 0.000,B 0.000,C 90.000,E1 104.828} C_DIS
LIN {X 0.103,Y -475.449,Z 439.358,A 0.000,B 0.000,C 90.000,E1 100.433} C_DIS
LIN {X -0.059,Y -476.098,Z 439.356,A 0.000,B 0.000,C 90.000,E1 100.141} C_DIS
LIN {X -0.256,Y -482.018,Z 439.331,A 0.000,B 0.000,C 90.000,E1 95.511} C_DIS
LIN {X -0.139,Y -482.864,Z 439.322,A 0.000,B 0.000,C 90.000,E1 93.955} C_DIS
LIN {X 0.015,Y -485.459,Z 439.305,A 0.000,B 0.000,C 90.000,E1 90.859} C_DIS
LIN {X -0.021,Y -485.500,Z 439.300,A 0.000,B 0.000,C 90.000,E1 89.943} C_DIS
LIN {X 0.047,Y -486.384,Z 439.281,A 0.000,B 0.000,C 90.000,E1 86.560} C_DIS
LIN {X -0.128,Y -486.365,Z 439.279,A 0.000,B 0.000,C 90.000,E1 86.274} C_DIS
LIN {X -0.039,Y -484.690,Z 439.254,A 0.000,B 0.000,C 90.000,E1 81.659} C_DIS
LIN {X 0.106,Y -484.062,Z 439.250,A 0.000,B 0.000,C 90.000,E1 81.027} C_DIS
LIN {X -0.129,Y -480.635,Z 439.228,A 0.000,B 0.000,C 90.000,E1 77.048} C_DIS
LIN {X 0.197,Y -480.330,Z 439.226,A 0.000,B 0.000,C 90.000,E1 76.700} C_DIS
LIN {X 0.100,Y -474.142,Z 439.200,A 0.000,B 0.000,C 90.000,E1 72.054} C_DIS
LIN {X -0.033,Y -465.618,Z 439.173,A 0.000,B 0.000,C 90.000,E1 67.050} C_DIS
LIN {X -0.079,Y -463.148,Z 439.167,A 0.000,B 0.000,C 90.000,E1 65.973} C_DIS
LIN {X -0.119,Y -463.144,Z 439.166,A 0.000,B 0.000,C 90.000,E1 65.973} C_DIS
LIN {X 0.015,Y -475.956,Z 439.157,A 0.000,B 0.000,C 90.000,E1 64.204} C_DIS
LIN {X 0.140,Y -484.939,Z 439.150,A 0.000,B 0.000,C 90.000,E1 62.948} C_DIS
LIN {X -0.071,Y -489.160,Z 439.146,A 0.000,B 0.000,C 90.000,E1 62.359} C_DIS
LIN {X -0.024,Y -494.054,Z 439.142,A 0.000,B 0.000,C 90.000,E1 61.591} C_DIS
LIN {X 0.033,Y -496.860,Z 439.140,A 0.000,B 0.000,C 90.000,E1 61.129} C_DIS
LIN {X -0.091,Y -500.325,Z 439.136,A 0.000,B 0.000,C 90.000,E1 60.539} C_DIS
LIN {X 0.062,Y -503.436,Z 439.133,A 0.000,B 0.000,C 90.000,E1 59.921} C_DIS
LIN {X -0.012,Y -506.224,Z 439.130,A 0.000,B 0.000,C 90.000,E1 59.331} C_DIS
LIN {X -0.068,Y -508.704,Z 439.126,A 0.000,B 0.000,C 90.000,E1 58.742} C_DIS
LIN {X 0.157,Y -510.873,Z 439.123,A 0.000,B 0.000,C 90.000,E1 58.122} C_DIS
LIN {X 0.125,Y -512.659,Z 439.120,A 0.000,B 0.000,C 90.000,E1 57.533} C_DIS
LIN {X 0.037,Y -513.486,Z 439.118,A 0.000,B 0.000,C 90.000,E1 57.248} C_DIS
LIN {X 0.302,Y -514.840,Z 439.115,A 0.000,B 0.000,C 90.000,E1 56.628} C_DIS
LIN {X -0.208,Y -516.459,Z 439.110,A 0.000,B 0.000,C 90.000,E1 55.801} C_DIS
LIN {X 0.016,Y -517.453,Z 439.105,A 0.000,B 0.000,C 90.000,E1 54.895} C_DIS
LIN {X 0.250,Y -517.973,Z 439.100,A 0.000,B 0.000,C 90.000,E1 53.989} C_DIS
LIN {X 0.010,Y -518.121,Z 439.094,A 0.000,B 0.000,C 90.000,E1 52.844} C_DIS
LIN {X -0.169,Y -518.020,Z 439.089,A 0.000,B 0.000,C 90.000,E1 51.984} C_DIS
LIN {X 0.031,Y -517.822,Z 439.085,A 0.000,B 0.000,C 90.000,E1 51.376} C_DIS
LIN {X 0.111,Y -517.028,Z 439.079,A 0.000,B 0.000,C 90.000,E1 50.194} C_DIS
LIN {X 0.172,Y -516.097,Z 439.072,A 0.000,B 0.000,C 90.000,E1 49.013} C_DIS
LIN {X 0.169,Y -514.939,Z 439.066,A 0.000,B 0.000,C 90.000,E1 47.838} C_DIS
LIN {X 0.065,Y -513.417,Z 439.058,A 0.000,B 0.000,C 90.000,E1 46.377} C_DIS
LIN {X 0.202,Y -510.537,Z 439.043,A 0.000,B 0.000,C 90.000,E1 43.704} C_DIS
LIN {X -0.223,Y -508.398,Z 439.031,A 0.000,B 0.000,C 90.000,E1 41.676} C_DIS
LIN {X 0.040,Y -507.160,Z 439.025,A 0.000,B 0.000,C 90.000,E1 40.458} C_DIS
LIN {X -0.038,Y -505.058,Z 439.013,A 0.000,B 0.000,C 90.000,E1 38.382} C_DIS
LIN {X 0.136,Y -503.534,Z 439.005,A 0.000,B 0.000,C 90.000,E1 36.870} C_DIS
LIN {X -0.197,Y -502.508,Z 439.000,A 0.000,B 0.000,C 90.000,E1 36.011} C_DIS
LIN {X 0.042,Y -500.780,Z 438.992,A 0.000,B 0.000,C 90.000,E1 34.485} C_DIS
LIN {X -0.038,Y -499.269,Z 438.985,A 0.000,B 0.000,C 90.000,E1 33.293} C_DIS
LIN {X 0.001,Y -497.708,Z 438.978,A 0.000,B 0.000,C 90.000,E1 32.084} C_DIS
LIN {X 0.022,Y -496.172,Z 438.972,A 0.000,B 0.000,C 90.000,E1 30.875} C_DIS
LIN {X -0.120,Y -493.734,Z 438.962,A 0.000,B 0.000,C 90.000,E1 29.077} C_DIS
LIN {X 0.119,Y -491.039,Z 438.950,A 0.000,B 0.000,C 90.000,E1 26.924} C_DIS
LIN {X -0.095,Y -487.660,Z 438.933,A 0.000,B 0.000,C 90.000,E1 23.898} C_DIS
LIN {X 0.289,Y -484.859,Z 438.914,A 0.000,B 0.000,C 90.000,E1 20.482} C_DIS
LIN {X 0.019,Y -483.459,Z 438.902,A 0.000,B 0.000,C 90.000,E1 18.362} C_DIS
LIN {X 0.182,Y -482.452,Z 438.894,A 0.000,B 0.000,C 90.000,E1 16.804} C_DIS
LIN {X 0.176,Y -481.161,Z 438.883,A 0.000,B 0.000,C 90.000,E1 14.954} C_DIS
LIN {X 0.000,Y -479.294,Z 438.866,A 0.000,B 0.000,C 90.000,E1 11.883} C_DIS
LIN {X -0.100,Y -478.487,Z 438.854,A 0.000,B 0.000,C 90.000,E1 9.726} C_DIS
LIN {X -0.210,Y -477.859,Z 438.839,A 0.000,B 0.000,C 90.000,E1 6.947} C_DIS
LIN {X -0.014,Y -477.967,Z 438.823,A 0.000,B 0.000,C 90.000,E1 4.131} C_DIS
LIN {X 0.054,Y -479.451,Z 438.802,A 0.000,B 0.000,C 90.000,E1 0.401} C_DIS
LIN {X -0.110,Y -480.687,Z 438.792,A 0.000,B 0.000,C 90.000,E1 358.568} C_DIS
LIN {X 0.233,Y -482.517,Z 438.782,A 0.000,B 0.000,C 90.000,E1 356.674} C_DIS
LIN {X -0.161,Y -486.811,Z 438.763,A 0.000,B 0.000,C 90.000,E1 353.337} C_DIS
LIN {X -0.107,Y -491.463,Z 438.746,A 0.000,B 0.000,C 90.000,E1 350.274} C_DIS
LIN {X -0.106,Y -497.460,Z 438.727,A 0.000,B 0.000,C 90.000,E1 346.937} C_DIS
LIN {X 0.039,Y -504.825,Z 438.709,A 0.000,B 0.000,C 90.000,E1 343.614} C_DIS
LIN {X 0.239,Y -511.504,Z 438.694,A 0.000,B 0.000,C 90.000,E1 340.913} C_DIS
LIN {X -0.244,Y -517.063,Z 438.683,A 0.000,B 0.000,C 90.000,E1 338.901} C_DIS
LIN {X 0.122,Y -521.827,Z 438.673,A 0.000,B 0.000,C 90.000,E1 337.102} C_DIS
LIN {X -0.049,Y -525.901,Z 438.665,A 0.000,B 0.000,C 90.000,E1 335.665} C_DIS
LIN {X -0.047,Y -531.550,Z 438.654,A 0.000,B 0.000,C 90.000,E1 333.640} C_DIS
LIN {X -0.146,Y -537.263,Z 438.642,A 0.000,B 0.000,C 90.000,E1 331.641} C_DIS
LIN {X -0.053,Y -541.478,Z 438.634,A 0.000,B 0.000,C 90.000,E1 330.205} C_DIS
LIN {X -0.080,Y -545.638,Z 438.627,A 0.000,B 0.000,C 90.000,E1 328.791} C_DIS
LIN {X -0.025,Y -549.780,Z 438.619,A 0.000,B 0.000,C 90.000,E1 327.375} C_DIS
LIN {X 0.226,Y -555.409,Z 438.608,A 0.000,B 0.000,C 90.000,E1 325.388} C_DIS
LIN {X -0.068,Y -560.340,Z 438.599,A 0.000,B 0.000,C 90.000,E1 323.749} C_DIS
LIN {X 0.190,Y -565.292,Z 438.589,A 0.000,B 0.000,C 90.000,E1 322.065} C_DIS
LIN {X -0.186,Y -572.315,Z 438.577,A 0.000,B 0.000,C 90.000,E1 319.908} C_DIS
LIN {X -0.140,Y -578.458,Z 438.567,A 0.000,B 0.000,C 90.000,E1 318.000} C_DIS
LIN {X -0.115,Y -583.585,Z 438.558,A 0.000,B 0.000,C 90.000,E1 316.377} C_DIS
LIN {X 0.341,Y -590.532,Z 438.546,A 0.000,B 0.000,C 90.000,E1 314.190} C_DIS
LIN {X -0.037,Y -596.661,Z 438.535,A 0.000,B 0.000,C 90.000,E1 312.366} C_DIS
LIN {X -0.021,Y -601.770,Z 438.527,A 0.000,B 0.000,C 90.000,E1 310.782} C_DIS
LIN {X 0.052,Y -605.101,Z 438.521,A 0.000,B 0.000,C 90.000,E1 309.725} C_DIS
LIN {X 0.059,Y -609.246,Z 438.514,A 0.000,B 0.000,C 90.000,E1 308.418} C_DIS
LIN {X -0.055,Y -613.865,Z 438.505,A 0.000,B 0.000,C 90.000,E1 306.870} C_DIS
LIN {X -0.271,Y -617.690,Z 438.498,A 0.000,B 0.000,C 90.000,E1 305.598} C_DIS
LIN {X 0.085,Y -621.304,Z 438.491,A 0.000,B 0.000,C 90.000,E1 304.278} C_DIS
LIN {X -0.018,Y -624.795,Z 438.483,A 0.000,B 0.000,C 90.000,E1 303.007} C_DIS
LIN {X 0.109,Y -628.107,Z 438.476,A 0.000,B 0.000,C 90.000,E1 301.720} C_DIS
LIN {X -0.008,Y -631.920,Z 438.468,A 0.000,B 0.000,C 90.000,E1 300.207} C_DIS
LIN {X -0.119,Y -634.338,Z 438.462,A 0.000,B 0.000,C 90.000,E1 299.205} C_DIS
LIN {X -0.117,Y -637.818,Z 438.454,A 0.000,B 0.000,C 90.000,E1 297.692} C_DIS
LIN {X 0.100,Y -640.098,Z 438.448,A 0.000,B 0.000,C 90.000,E1 296.668} C_DIS
LIN {X 0.071,Y -642.255,Z 438.443,A 0.000,B 0.000,C 90.000,E1 295.668} C_DIS
LIN {X 0.426,Y -644.756,Z 438.436,A 0.000,B 0.000,C 90.000,E1 294.387} C_DIS
LIN {X -0.304,Y -647.131,Z 438.429,A 0.000,B 0.000,C 90.000,E1 293.206} C_DIS
LIN {X -0.311,Y -649.589,Z 438.421,A 0.000,B 0.000,C 90.000,E1 291.716} C_DIS
LIN {X 0.244,Y -651.513,Z 438.414,A 0.000,B 0.000,C 90.000,E1 290.429} C_DIS
LIN {X 0.131,Y -653.004,Z 438.408,A 0.000,B 0.000,C 90.000,E1 289.450} C_DIS
LIN {X -0.097,Y -654.547,Z 438.401,A 0.000,B 0.000,C 90.000,E1 288.236} C_DIS
LIN {X 0.240,Y -655.610,Z 438.396,A 0.000,B 0.000,C 90.000,E1 287.221} C_DIS
LIN {X -0.146,Y -656.731,Z 438.389,A 0.000,B 0.000,C 90.000,E1 286.024} C_DIS
LIN {X 0.113,Y -657.547,Z 438.382,A 0.000,B 0.000,C 90.000,E1 284.773} C_DIS
LIN {X 0.219,Y -658.163,Z 438.375,A 0.000,B 0.000,C 90.000,E1 283.536} C_DIS
LIN {X -0.307,Y -658.651,Z 438.369,A 0.000,B 0.000,C 90.000,E1 282.355} C_DIS
LIN {X 0.106,Y -658.740,Z 438.359,A 0.000,B 0.000,C 90.000,E1 280.602} C_DIS
LIN {X 0.086,Y -658.543,Z 438.352,A 0.000,B 0.000,C 90.000,E1 279.378} C_DIS
LIN {X 0.073,Y -658.145,Z 438.347,A 0.000,B 0.000,C 90.000,E1 278.398} C_DIS
LIN {X -0.059,Y -657.373,Z 438.340,A 0.000,B 0.000,C 90.000,E1 277.182} C_DIS
LIN {X -0.078,Y -656.509,Z 438.334,A 0.000,B 0.000,C 90.000,E1 276.201} C_DIS
LIN {X 0.030,Y -655.663,Z 438.330,A 0.000,B 0.000,C 90.000,E1 275.454} C_DIS
LIN {X 0.188,Y -654.766,Z 438.326,A 0.000,B 0.000,C 90.000,E1 274.702} C_DIS
LIN {X -0.135,Y -652.846,Z 438.319,A 0.000,B 0.000,C 90.000,E1 273.498} C_DIS
LIN {X 0.170,Y -650.695,Z 438.313,A 0.000,B 0.000,C 90.000,E1 272.236} C_DIS
LIN {X -0.215,Y -648.266,Z 438.306,A 0.000,B 0.000,C 90.000,E1 271.031} C_DIS
LIN {X 0.213,Y -646.111,Z 438.300,A 0.000,B 0.000,C 90.000,E1 270.000} C_DIS
LIN {X -0.033,Y -643.830,Z 438.295,A 0.000,B 0.000,C 90.000,E1 269.026} C_DIS
LIN {X 0.113,Y -640.692,Z 438.288,A 0.000,B 0.000,C 90.000,E1 267.764} C_DIS
LIN {X -0.181,Y -638.024,Z 438.282,A 0.000,B 0.000,C 90.000,E1 266.788} C_DIS
LIN {X 0.238,Y -633.869,Z 438.274,A 0.000,B 0.000,C 90.000,E1 265.241} C_DIS
LIN {X 0.254,Y -630.374,Z 438.267,A 0.000,B 0.000,C 90.000,E1 263.976} C_DIS
LIN {X 0.281,Y -626.755,Z 438.260,A 0.000,B 0.000,C 90.000,E1 262.704} C_DIS
LIN {X -0.143,Y -623.813,Z 438.254,A 0.000,B 0.000,C 90.000,E1 261.724} C_DIS
LIN {X -0.126,Y -620.023,Z 438.247,A 0.000,B 0.000,C 90.000,E1 260.443} C_DIS
LIN {X -0.029,Y -614.580,Z 438.237,A 0.000,B 0.000,C 90.000,E1 258.634} C_DIS
LIN {X 0.178,Y -609.692,Z 438.228,A 0.000,B 0.000,C 90.000,E1 257.061} C_DIS
LIN {X 0.224,Y -605.485,Z 438.221,A 0.000,B 0.000,C 90.000,E1 255.755} C_DIS
LIN {X -0.068,Y -600.228,Z 438.212,A 0.000,B 0.000,C 90.000,E1 254.212} C_DIS
LIN {X 0.115,Y -596.672,Z 438.206,A 0.000,B 0.000,C 90.000,E1 253.142} C_DIS
LIN {X 0.115,Y -592.124,Z 438.199,A 0.000,B 0.000,C 90.000,E1 251.819} C_DIS
LIN {X 0.031,Y -587.498,Z 438.192,A 0.000,B 0.000,C 90.000,E1 250.496} C_DIS
LIN {X 0.056,Y -582.712,Z 438.184,A 0.000,B 0.000,C 90.000,E1 249.156} C_DIS
LIN {X -0.182,Y -578.728,Z 438.178,A 0.000,B 0.000,C 90.000,E1 248.103} C_DIS
LIN {X 0.060,Y -574.670,Z 438.172,A 0.000,B 0.000,C 90.000,E1 246.997} C_DIS
LIN {X -0.227,Y -569.366,Z 438.165,A 0.000,B 0.000,C 90.000,E1 245.665} C_DIS
LIN {X 0.104,Y -565.093,Z 438.159,A 0.000,B 0.000,C 90.000,E1 244.537} C_DIS
LIN {X 0.212,Y -558.577,Z 438.149,A 0.000,B 0.000,C 90.000,E1 242.871} C_DIS
LIN {X -0.312,Y -552.099,Z 438.140,A 0.000,B 0.000,C 90.000,E1 241.257} C_DIS
LIN {X 0.043,Y -545.776,Z 438.131,A 0.000,B 0.000,C 90.000,E1 239.537} C_DIS
LIN {X -0.208,Y -539.539,Z 438.121,A 0.000,B 0.000,C 90.000,E1 237.867} C_DIS
LIN {X -0.010,Y -534.370,Z 438.113,A 0.000,B 0.000,C 90.000,E1 236.421} C_DIS
LIN {X 0.055,Y -527.094,Z 438.102,A 0.000,B 0.000,C 90.000,E1 234.402} C_DIS
LIN {X -0.095,Y -522.064,Z 438.094,A 0.000,B 0.000,C 90.000,E1 232.970} C_DIS
LIN {X 0.070,Y -517.113,Z 438.086,A 0.000,B 0.000,C 90.000,E1 231.492} C_DIS
LIN {X 0.107,Y -507.015,Z 438.068,A 0.000,B 0.000,C 90.000,E1 228.243} C_DIS
LIN {X 0.066,Y -501.812,Z 438.058,A 0.000,B 0.000,C 90.000,E1 226.458} C_DIS
LIN {X 0.090,Y -495.889,Z 438.047,A 0.000,B 0.000,C 90.000,E1 224.352} C_DIS
LIN {X 0.145,Y -489.261,Z 438.033,A 0.000,B 0.000,C 90.000,E1 221.919} C_DIS
LIN {X 0.081,Y -484.455,Z 438.023,A 0.000,B 0.000,C 90.000,E1 220.092} C_DIS
LIN {X -0.026,Y -479.850,Z 438.013,A 0.000,B 0.000,C 90.000,E1 218.257} C_DIS
LIN {X 0.179,Y -473.210,Z 437.997,A 0.000,B 0.000,C 90.000,E1 215.438} C_DIS
LIN {X 0.023,Y -469.062,Z 437.987,A 0.000,B 0.000,C 90.000,E1 213.579} C_DIS
LIN {X 0.169,Y -464.980,Z 437.976,A 0.000,B 0.000,C 90.000,E1 211.671} C_DIS
LIN {X -0.027,Y -460.955,Z 437.966,A 0.000,B 0.000,C 90.000,E1 209.795} C_DIS
LIN {X -0.260,Y -457.628,Z 437.957,A 0.000,B 0.000,C 90.000,E1 208.231} C_DIS
LIN {X -0.149,Y -454.268,Z 437.948,A 0.000,B 0.000,C 90.000,E1 206.616} C_DIS
